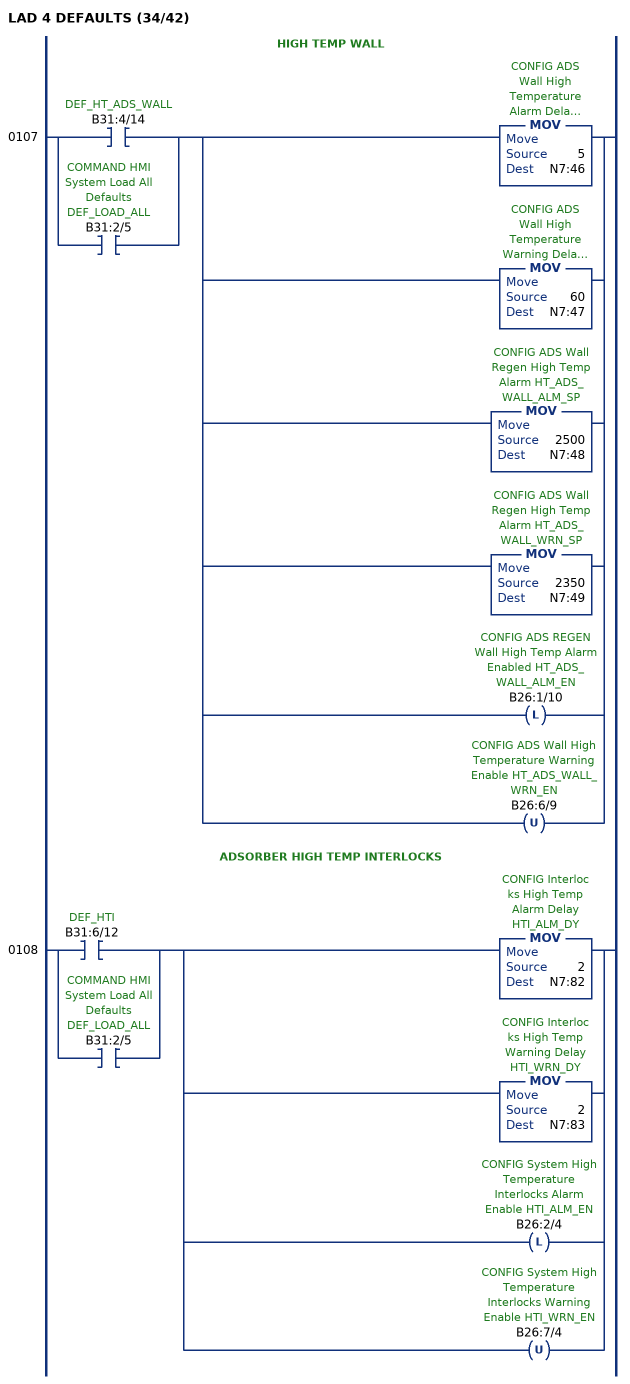
% Rung: 107 %
% TITLE: HIGH TEMP WALL %
SOR BST XIC B31:4/14 NXB XIC B31:2/5 BND BST MOV 5 N7:46 NXB MOV 60 N7:47 NXB MOV 2500 N7:48 NXB MOV 2350 N7:49 NXB OTL B26:1/10 NXB OTU B26:6/9 BND EOR
%   B31:4/14  DEF_HT_ADS_WALL %
%   B31:2/5  DEF_LOAD_ALL  "COMMAND HMI System Load All Defaults" %
%   N7:46  HT_ADS_WALL_ALM_DLY  "CONFIG ADS Wall High Temperature Alarm Delay" %
%   N7:47  HT_ADS_WALL_WRN_DLY  "CONFIG ADS Wall High Temperature Warning Delay" %
%   N7:48  HT_ADS_WALL_ALM_SP  "CONFIG ADS Wall Regen High Temp Alarm" %
%   N7:49  HT_ADS_WALL_WRN_SP  "CONFIG ADS Wall Regen High Temp Alarm" %
%   B26:1/10  HT_ADS_WALL_ALM_EN  "CONFIG ADS REGEN Wall High Temp Alarm Enabled" %
%   B26:6/9  HT_ADS_WALL_WRN_EN  "CONFIG ADS Wall High Temperature Warning Enable" %
% Rung: 108 %
% TITLE: ADSORBER HIGH TEMP INTERLOCKS %
SOR BST XIC B31:6/12 NXB XIC B31:2/5 BND BST MOV 2 N7:82 NXB MOV 2 N7:83 NXB OTL B26:2/4 NXB OTU B26:7/4 BND EOR
%   B31:6/12  DEF_HTI %
%   B31:2/5  DEF_LOAD_ALL  "COMMAND HMI System Load All Defaults" %
%   N7:82  HTI_ALM_DY  "CONFIG Interlocks High Temp Alarm Delay" %
%   N7:83  HTI_WRN_DY  "CONFIG Interlocks High Temp Warning Delay" %
%   B26:2/4  HTI_ALM_EN  "CONFIG System High Temperature Interlocks Alarm Enable" %
%   B26:7/4  HTI_WRN_EN  "CONFIG System High Temperature Interlocks Warning Enable" %

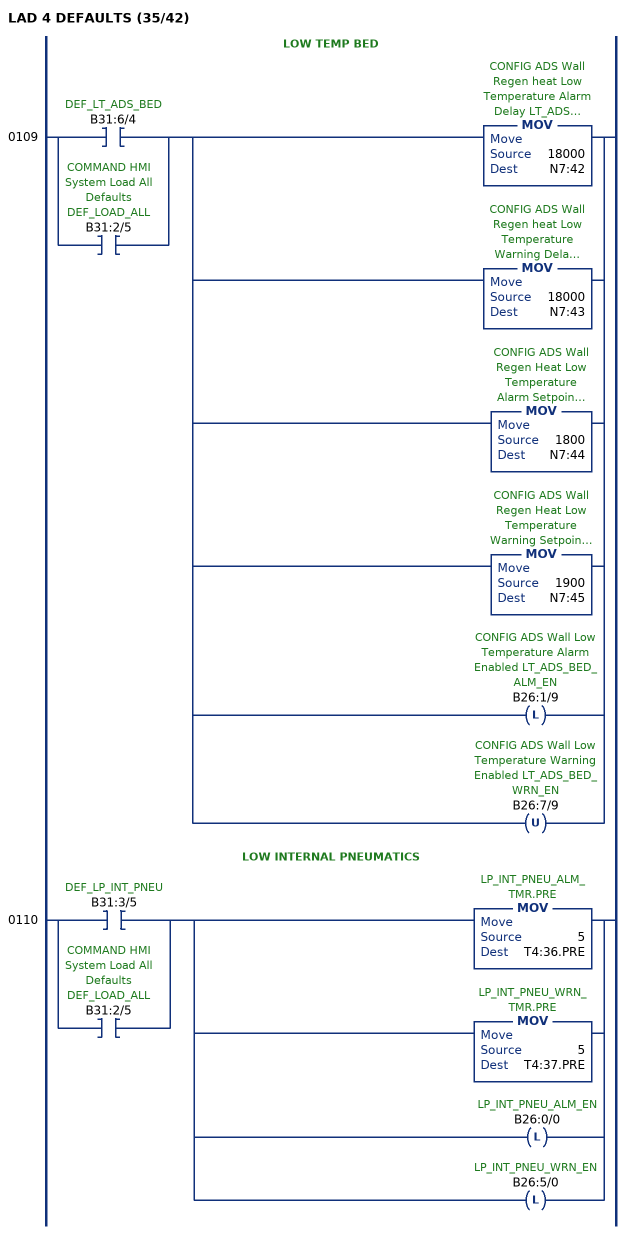
% Rung: 109 %
% TITLE: LOW TEMP BED %
SOR BST XIC B31:6/4 NXB XIC B31:2/5 BND BST MOV 18000 N7:42 NXB MOV 18000 N7:43 NXB MOV 1800 N7:44 NXB MOV 1900 N7:45 NXB OTL B26:1/9 NXB OTU B26:7/9 BND EOR
%   B31:6/4  DEF_LT_ADS_BED %
%   B31:2/5  DEF_LOAD_ALL  "COMMAND HMI System Load All Defaults" %
%   N7:42  LT_ADS_BED_ALM_DLY  "CONFIG ADS Wall Regen heat Low Temperature Alarm Delay" %
%   N7:43  LT_ADS_BED_WRN_DLY  "CONFIG ADS Wall Regen heat Low Temperature Warning Delay" %
%   N7:44  LT_ADS_BED_ALM_SP  "CONFIG ADS Wall Regen Heat Low Temperature Alarm Setpoint" %
%   N7:45  LT_ADS_BED_WRN_SP  "CONFIG ADS Wall Regen Heat Low Temperature Warning Setpoint" %
%   B26:1/9  LT_ADS_BED_ALM_EN  "CONFIG ADS Wall Low Temperature Alarm Enabled" %
%   B26:7/9  LT_ADS_BED_WRN_EN  "CONFIG ADS Wall Low Temperature Warning Enabled" %
% Rung: 110 %
% TITLE: LOW INTERNAL PNEUMATICS %
SOR BST XIC B31:3/5 NXB XIC B31:2/5 BND BST MOV 5 T4:36.PRE NXB MOV 5 T4:37.PRE NXB OTL B26:0/0 NXB OTL B26:5/0 BND EOR
%   B31:3/5  DEF_LP_INT_PNEU %
%   B31:2/5  DEF_LOAD_ALL  "COMMAND HMI System Load All Defaults" %
%   T4:36  LP_INT_PNEU_ALM_TMR %
%   T4:37  LP_INT_PNEU_WRN_TMR %
%   B26:0/0  LP_INT_PNEU_ALM_EN %
%   B26:5/0  LP_INT_PNEU_WRN_EN %

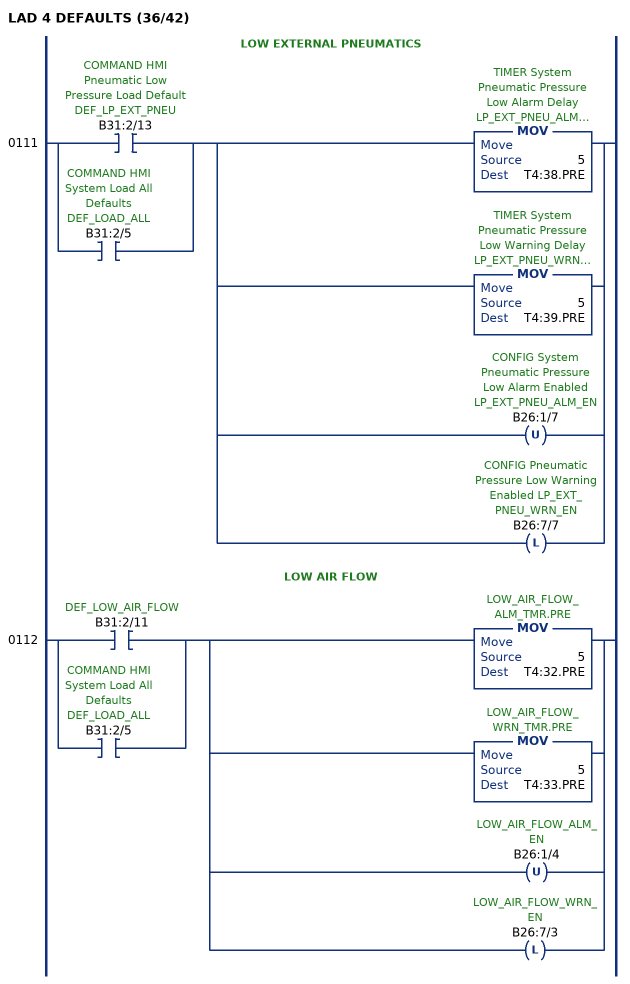
% Rung: 111 %
% TITLE: LOW EXTERNAL PNEUMATICS %
SOR BST XIC B31:2/13 NXB XIC B31:2/5 BND BST MOV 5 T4:38.PRE NXB MOV 5 T4:39.PRE NXB OTU B26:1/7 NXB OTL B26:7/7 BND EOR
%   B31:2/13  DEF_LP_EXT_PNEU  "COMMAND HMI Pneumatic Low Pressure Load Default" %
%   B31:2/5  DEF_LOAD_ALL  "COMMAND HMI System Load All Defaults" %
%   T4:38  LP_EXT_PNEU_ALM_TMR  "TIMER System Pneumatic Pressure Low Alarm Delay" %
%   T4:39  LP_EXT_PNEU_WRN_TMR  "TIMER System Pneumatic Pressure Low Warning Delay" %
%   B26:1/7  LP_EXT_PNEU_ALM_EN  "CONFIG System Pneumatic Pressure Low Alarm Enabled" %
%   B26:7/7  LP_EXT_PNEU_WRN_EN  "CONFIG Pneumatic Pressure Low Warning Enabled" %
% Rung: 112 %
% TITLE: LOW AIR FLOW %
SOR BST XIC B31:2/11 NXB XIC B31:2/5 BND BST MOV 5 T4:32.PRE NXB MOV 5 T4:33.PRE NXB OTU B26:1/4 NXB OTL B26:7/3 BND EOR
%   B31:2/11  DEF_LOW_AIR_FLOW %
%   B31:2/5  DEF_LOAD_ALL  "COMMAND HMI System Load All Defaults" %
%   T4:32  LOW_AIR_FLOW_ALM_TMR %
%   T4:33  LOW_AIR_FLOW_WRN_TMR %
%   B26:1/4  LOW_AIR_FLOW_ALM_EN %
%   B26:7/3  LOW_AIR_FLOW_WRN_EN %

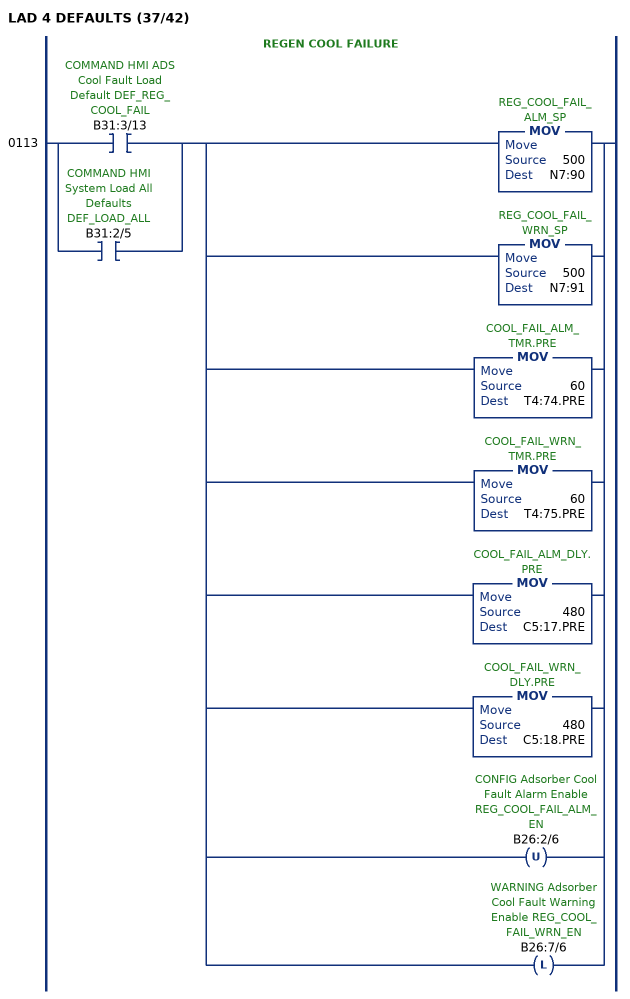
% Rung: 113 %
% TITLE: REGEN COOL FAILURE %
SOR BST XIC B31:3/13 NXB XIC B31:2/5 BND BST MOV 500 N7:90 NXB MOV 500 N7:91 NXB MOV 60 T4:74.PRE NXB MOV 60 T4:75.PRE NXB MOV 480 C5:17.PRE NXB MOV 480 C5:18.PRE NXB OTU B26:2/6 NXB OTL B26:7/6 BND EOR
%   B31:3/13  DEF_REG_COOL_FAIL  "COMMAND HMI ADS Cool Fault Load Default" %
%   B31:2/5  DEF_LOAD_ALL  "COMMAND HMI System Load All Defaults" %
%   N7:90  REG_COOL_FAIL_ALM_SP %
%   N7:91  REG_COOL_FAIL_WRN_SP %
%   T4:74  COOL_FAIL_ALM_TMR %
%   T4:75  COOL_FAIL_WRN_TMR %
%   C5:17  COOL_FAIL_ALM_DLY %
%   C5:18  COOL_FAIL_WRN_DLY %
%   B26:2/6  REG_COOL_FAIL_ALM_EN  "CONFIG Adsorber Cool Fault Alarm Enable" %
%   B26:7/6  REG_COOL_FAIL_WRN_EN  "WARNING Adsorber Cool Fault Warning Enable" %

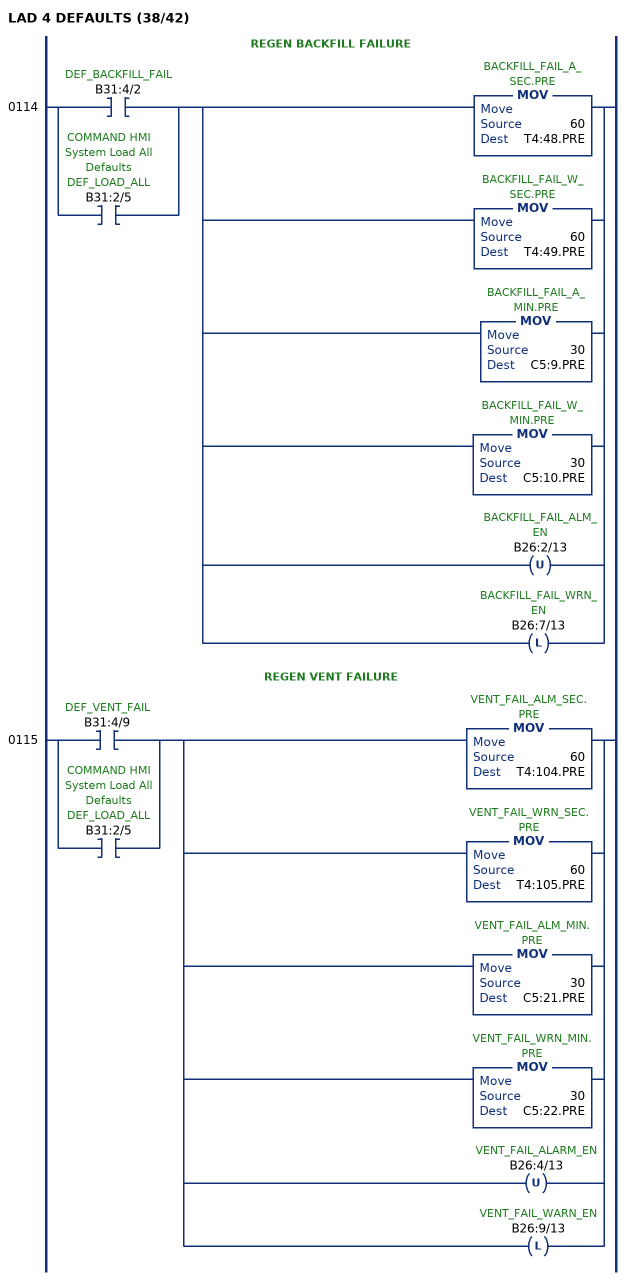
% Rung: 114 %
% TITLE: REGEN BACKFILL FAILURE %
SOR BST XIC B31:4/2 NXB XIC B31:2/5 BND BST MOV 60 T4:48.PRE NXB MOV 60 T4:49.PRE NXB MOV 30 C5:9.PRE NXB MOV 30 C5:10.PRE NXB OTU B26:2/13 NXB OTL B26:7/13 BND EOR
%   B31:4/2  DEF_BACKFILL_FAIL %
%   B31:2/5  DEF_LOAD_ALL  "COMMAND HMI System Load All Defaults" %
%   T4:48  BACKFILL_FAIL_A_SEC %
%   T4:49  BACKFILL_FAIL_W_SEC %
%   C5:9  BACKFILL_FAIL_A_MIN %
%   C5:10  BACKFILL_FAIL_W_MIN %
%   B26:2/13  BACKFILL_FAIL_ALM_EN %
%   B26:7/13  BACKFILL_FAIL_WRN_EN %
% Rung: 115 %
% TITLE: REGEN VENT FAILURE %
SOR BST XIC B31:4/9 NXB XIC B31:2/5 BND BST MOV 60 T4:104.PRE NXB MOV 60 T4:105.PRE NXB MOV 30 C5:21.PRE NXB MOV 30 C5:22.PRE NXB OTU B26:4/13 NXB OTL B26:9/13 BND EOR
%   B31:4/9  DEF_VENT_FAIL %
%   B31:2/5  DEF_LOAD_ALL  "COMMAND HMI System Load All Defaults" %
%   T4:104  VENT_FAIL_ALM_SEC %
%   T4:105  VENT_FAIL_WRN_SEC %
%   C5:21  VENT_FAIL_ALM_MIN %
%   C5:22  VENT_FAIL_WRN_MIN %
%   B26:4/13  VENT_FAIL_ALARM_EN %
%   B26:9/13  VENT_FAIL_WARN_EN %

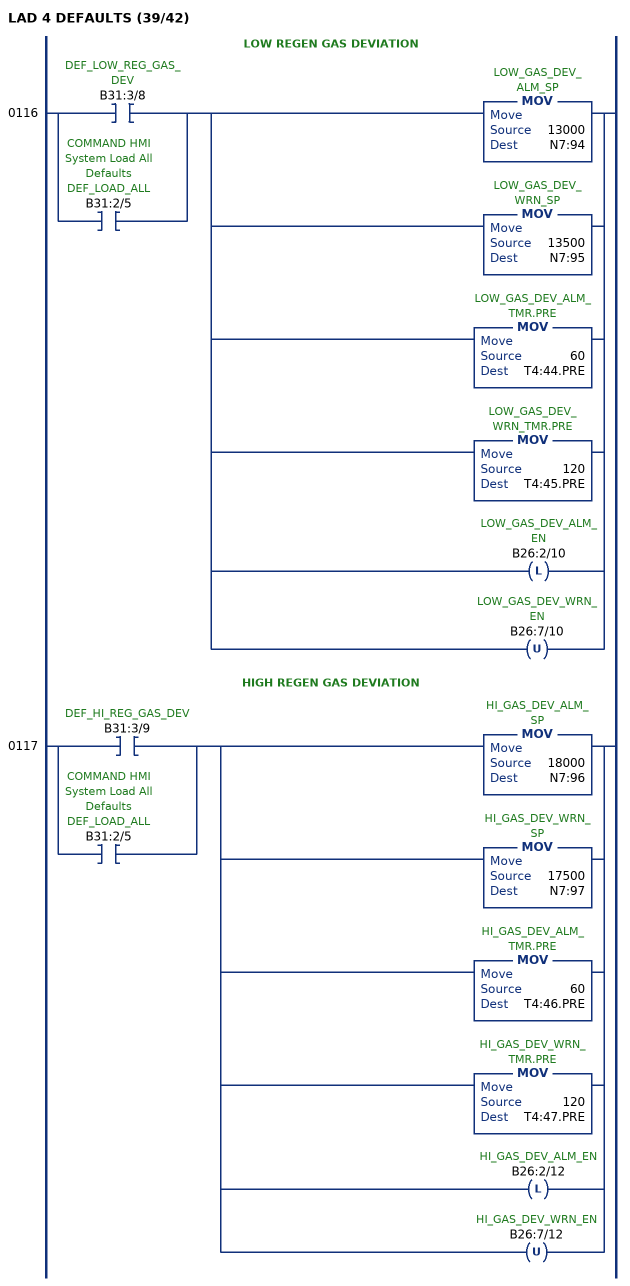
% Rung: 116 %
% TITLE: LOW REGEN GAS DEVIATION %
SOR BST XIC B31:3/8 NXB XIC B31:2/5 BND BST MOV 13000 N7:94 NXB MOV 13500 N7:95 NXB MOV 60 T4:44.PRE NXB MOV 120 T4:45.PRE NXB OTL B26:2/10 NXB OTU B26:7/10 BND EOR
%   B31:3/8  DEF_LOW_REG_GAS_DEV %
%   B31:2/5  DEF_LOAD_ALL  "COMMAND HMI System Load All Defaults" %
%   N7:94  LOW_GAS_DEV_ALM_SP %
%   N7:95  LOW_GAS_DEV_WRN_SP %
%   T4:44  LOW_GAS_DEV_ALM_TMR %
%   T4:45  LOW_GAS_DEV_WRN_TMR %
%   B26:2/10  LOW_GAS_DEV_ALM_EN %
%   B26:7/10  LOW_GAS_DEV_WRN_EN %
% Rung: 117 %
% TITLE: HIGH REGEN GAS DEVIATION %
SOR BST XIC B31:3/9 NXB XIC B31:2/5 BND BST MOV 18000 N7:96 NXB MOV 17500 N7:97 NXB MOV 60 T4:46.PRE NXB MOV 120 T4:47.PRE NXB OTL B26:2/12 NXB OTU B26:7/12 BND EOR
%   B31:3/9  DEF_HI_REG_GAS_DEV %
%   B31:2/5  DEF_LOAD_ALL  "COMMAND HMI System Load All Defaults" %
%   N7:96  HI_GAS_DEV_ALM_SP %
%   N7:97  HI_GAS_DEV_WRN_SP %
%   T4:46  HI_GAS_DEV_ALM_TMR %
%   T4:47  HI_GAS_DEV_WRN_TMR %
%   B26:2/12  HI_GAS_DEV_ALM_EN %
%   B26:7/12  HI_GAS_DEV_WRN_EN %

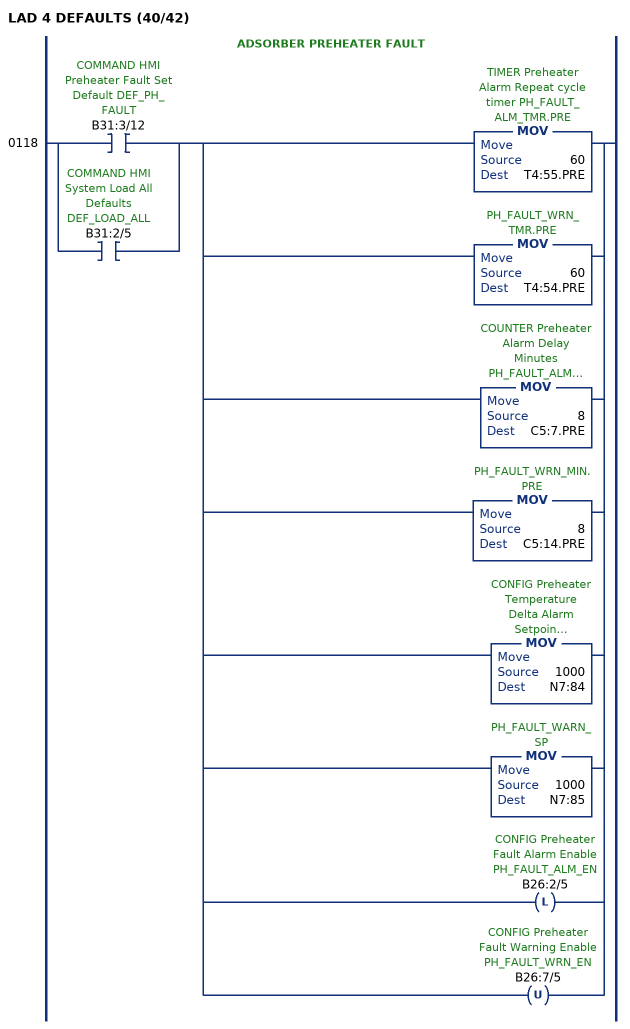
% Rung: 118 %
% TITLE: ADSORBER PREHEATER FAULT %
SOR BST XIC B31:3/12 NXB XIC B31:2/5 BND BST MOV 60 T4:55.PRE NXB MOV 60 T4:54.PRE NXB MOV 8 C5:7.PRE NXB MOV 8 C5:14.PRE NXB MOV 1000 N7:84 NXB MOV 1000 N7:85 NXB OTL B26:2/5 NXB OTU B26:7/5 BND EOR
%   B31:3/12  DEF_PH_FAULT  "COMMAND HMI Preheater Fault Set Default" %
%   B31:2/5  DEF_LOAD_ALL  "COMMAND HMI System Load All Defaults" %
%   T4:55  PH_FAULT_ALM_TMR  "TIMER Preheater Alarm Repeat cycle timer" %
%   T4:54  PH_FAULT_WRN_TMR %
%   C5:7  PH_FAULT_ALM_MIN  "COUNTER Preheater Alarm Delay Minutes" %
%   C5:14  PH_FAULT_WRN_MIN %
%   N7:84  PH_FAULT_ALARM_SP  "CONFIG Preheater Temperature Delta Alarm Setpoint" %
%   N7:85  PH_FAULT_WARN_SP %
%   B26:2/5  PH_FAULT_ALM_EN  "CONFIG Preheater Fault Alarm Enable" %
%   B26:7/5  PH_FAULT_WRN_EN  "CONFIG Preheater Fault Warning Enable" %

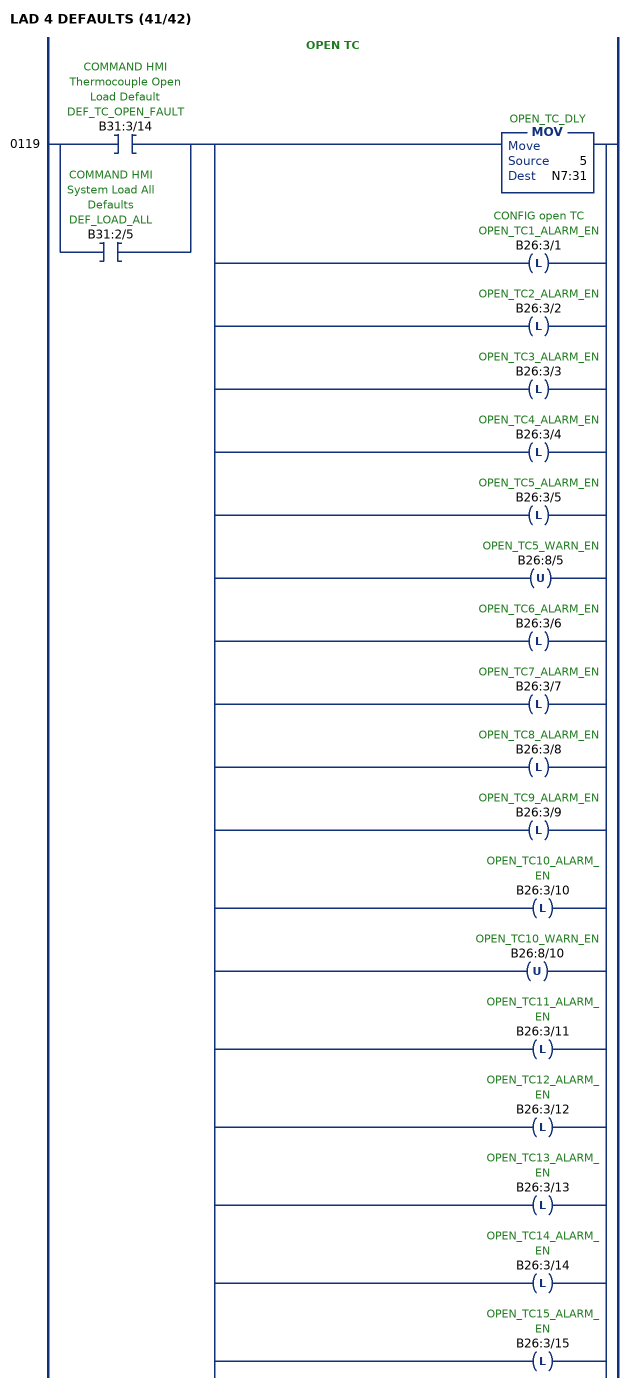

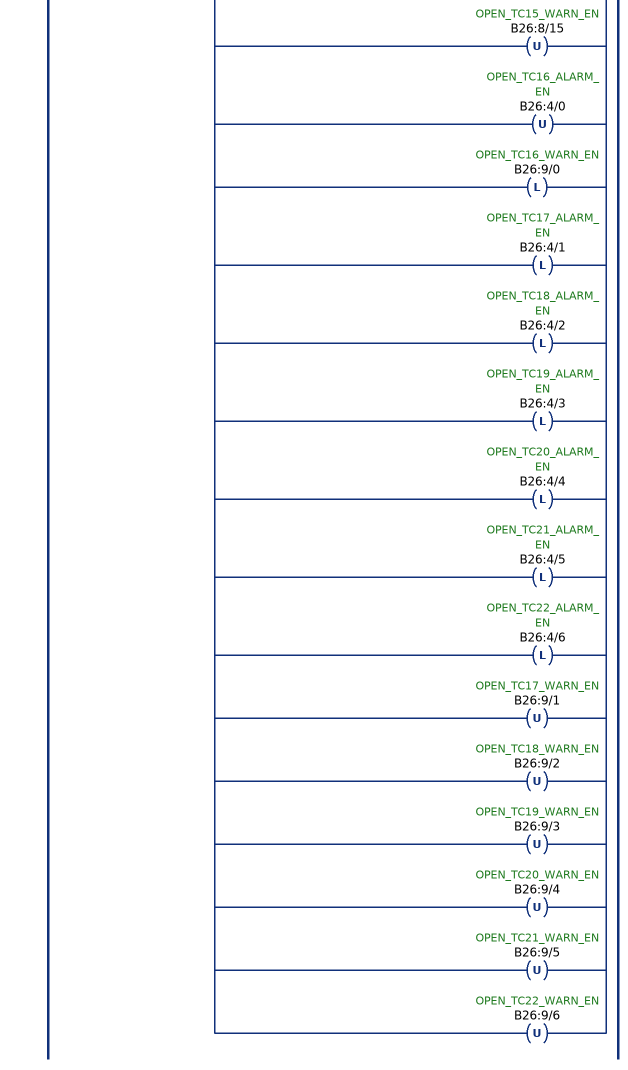
% Rung: 119 %
% TITLE: OPEN TC %
SOR BST XIC B31:3/14 NXB XIC B31:2/5 BND BST MOV 5 N7:31 NXB BST OTL B26:3/1 NXB OTL B26:3/2 NXB OTL B26:3/3 NXB OTL B26:3/4 NXB OTL B26:3/5 NXB OTU B26:8/5 BND NXB BST OTL B26:3/6 NXB OTL B26:3/7 NXB OTL B26:3/8 NXB OTL B26:3/9 NXB OTL B26:3/10 NXB OTU B26:8/10 BND NXB BST OTL B26:3/11 NXB OTL B26:3/12 NXB OTL B26:3/13 NXB OTL B26:3/14 NXB OTL B26:3/15 NXB OTU B26:8/15 BND NXB BST OTU B26:4/0 NXB OTL B26:9/0 BND NXB BST OTL B26:4/1 NXB OTL B26:4/2 NXB OTL B26:4/3 NXB OTL B26:4/4 NXB OTL B26:4/5 NXB OTL B26:4/6 BND NXB BST OTU B26:9/1 NXB OTU B26:9/2 NXB OTU B26:9/3 NXB OTU B26:9/4 NXB OTU B26:9/5 NXB OTU B26:9/6 BND BND EOR
%   B31:3/14  DEF_TC_OPEN_FAULT  "COMMAND HMI Thermocouple Open Load Default" %
%   B31:2/5  DEF_LOAD_ALL  "COMMAND HMI System Load All Defaults" %
%   N7:31  OPEN_TC_DLY %
%   B26:3/1  OPEN_TC1_ALARM_EN  "CONFIG open TC" %
%   B26:3/2  OPEN_TC2_ALARM_EN %
%   B26:3/3  OPEN_TC3_ALARM_EN %
%   B26:3/4  OPEN_TC4_ALARM_EN %
%   B26:3/5  OPEN_TC5_ALARM_EN %
%   B26:8/5  OPEN_TC5_WARN_EN %
%   B26:3/6  OPEN_TC6_ALARM_EN %
%   B26:3/7  OPEN_TC7_ALARM_EN %
%   B26:3/8  OPEN_TC8_ALARM_EN %
%   B26:3/9  OPEN_TC9_ALARM_EN %
%   B26:3/10  OPEN_TC10_ALARM_EN %
%   B26:8/10  OPEN_TC10_WARN_EN %
%   B26:3/11  OPEN_TC11_ALARM_EN %
%   B26:3/12  OPEN_TC12_ALARM_EN %
%   B26:3/13  OPEN_TC13_ALARM_EN %
%   B26:3/14  OPEN_TC14_ALARM_EN %
%   B26:3/15  OPEN_TC15_ALARM_EN %
%   B26:8/15  OPEN_TC15_WARN_EN %
%   B26:4/0  OPEN_TC16_ALARM_EN %
%   B26:9/0  OPEN_TC16_WARN_EN %
%   B26:4/1  OPEN_TC17_ALARM_EN %
%   B26:4/2  OPEN_TC18_ALARM_EN %
%   B26:4/3  OPEN_TC19_ALARM_EN %
%   B26:4/4  OPEN_TC20_ALARM_EN %
%   B26:4/5  OPEN_TC21_ALARM_EN %
%   B26:4/6  OPEN_TC22_ALARM_EN %
%   B26:9/1  OPEN_TC17_WARN_EN %
%   B26:9/2  OPEN_TC18_WARN_EN %
%   B26:9/3  OPEN_TC19_WARN_EN %
%   B26:9/4  OPEN_TC20_WARN_EN %
%   B26:9/5  OPEN_TC21_WARN_EN %
%   B26:9/6  OPEN_TC22_WARN_EN %

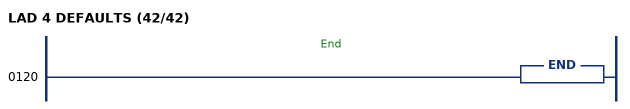
% Rung: 120 %
% End %
SOR END EOR

LADDER 5 "SYS_FAULTS"    % Monitors the system fault conditions %
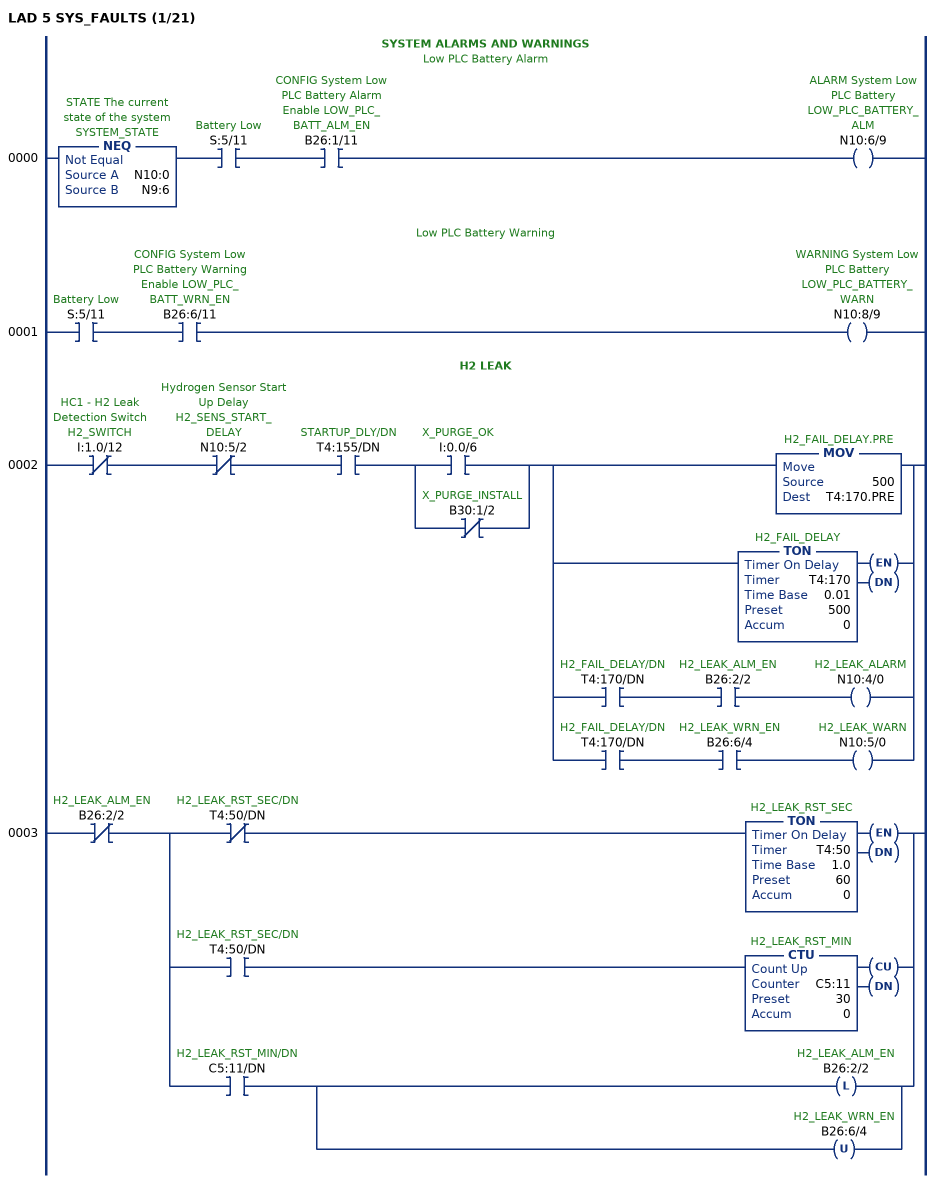
% Rung: 0 %
% TITLE: SYSTEM ALARMS AND WARNINGS %
% Low PLC Battery Alarm %
SOR NEQ N10:0 N9:6 XIC S:5/11 XIC B26:1/11 OTE N10:6/9 EOR
%   N10:0  SYSTEM_STATE  "STATE The current state of the system" %
%   N9:6  SYSTEM_PURGE %
%   S:5/11  "Battery Low" %
%   B26:1/11  LOW_PLC_BATT_ALM_EN  "CONFIG System Low PLC Battery Alarm Enable" %
%   N10:6/9  LOW_PLC_BATTERY_ALM  "ALARM System Low PLC Battery" %
% Rung: 1 %
% Low PLC Battery Warning %
SOR XIC S:5/11 XIC B26:6/11 OTE N10:8/9 EOR
%   S:5/11  "Battery Low" %
%   B26:6/11  LOW_PLC_BATT_WRN_EN  "CONFIG System Low PLC Battery Warning Enable" %
%   N10:8/9  LOW_PLC_BATTERY_WARN  "WARNING System Low PLC Battery" %
% Rung: 2 %
% TITLE: H2 LEAK %
SOR XIO I:1.0/12 XIO N10:5/2 XIC T4:155/DN BST XIC I:0.0/6 NXB XIO B30:1/2 BND BST MOV 500 T4:170.PRE NXB TON T4:170 0.01 500 0 NXB XIC T4:170/DN XIC B26:2/2 OTE N10:4/0 NXB XIC T4:170/DN XIC B26:6/4 OTE N10:5/0 BND EOR
%   I:1.0/12  H2_SWITCH  "HC1 - H2 Leak Detection Switch" %
%   N10:5/2  H2_SENS_START_DELAY  "Hydrogen Sensor Start Up Delay" %
%   T4:155  STARTUP_DLY %
%   I:0.0/6  X_PURGE_OK %
%   B30:1/2  X_PURGE_INSTALL %
%   T4:170  H2_FAIL_DELAY %
%   B26:2/2  H2_LEAK_ALM_EN %
%   N10:4/0  H2_LEAK_ALARM %
%   B26:6/4  H2_LEAK_WRN_EN %
%   N10:5/0  H2_LEAK_WARN %
% Rung: 3 %
SOR XIO B26:2/2 BST XIO T4:50/DN TON T4:50 1.0 60 0 NXB XIC T4:50/DN CTU C5:11 30 0 NXB XIC C5:11/DN BST OTL B26:2/2 NXB OTU B26:6/4 BND BND EOR
%   B26:2/2  H2_LEAK_ALM_EN %
%   T4:50  H2_LEAK_RST_SEC %
%   C5:11  H2_LEAK_RST_MIN %
%   B26:6/4  H2_LEAK_WRN_EN %

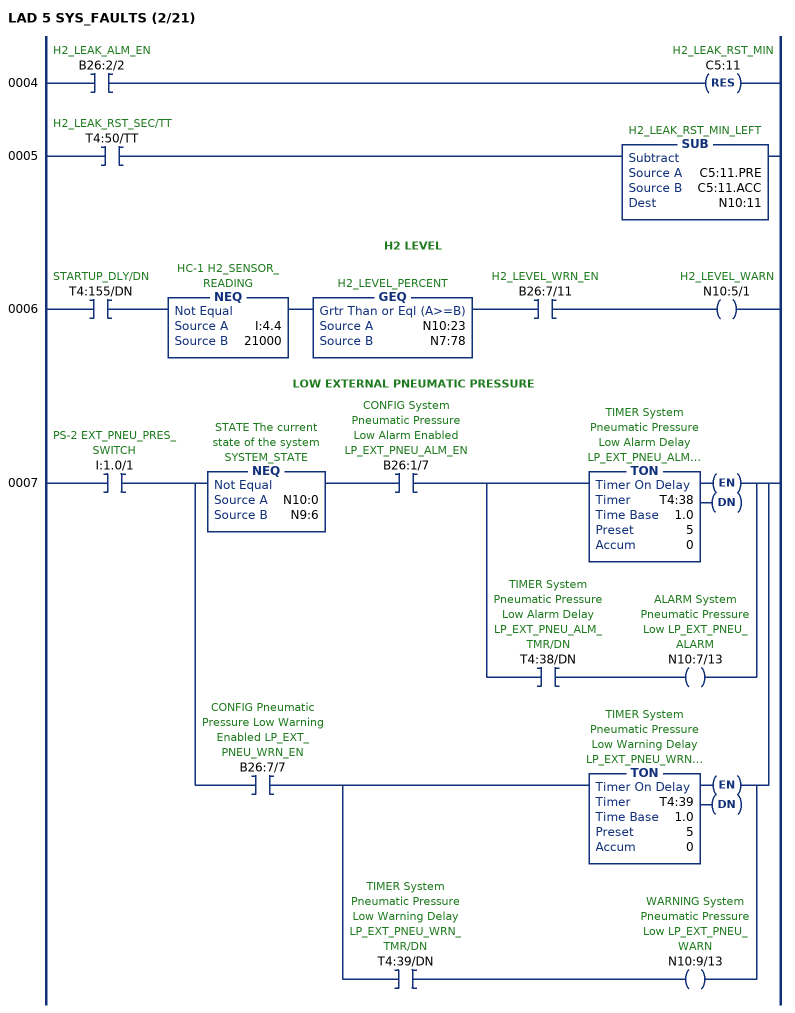
% Rung: 4 %
SOR XIC B26:2/2 RES C5:11 EOR
%   B26:2/2  H2_LEAK_ALM_EN %
%   C5:11  H2_LEAK_RST_MIN %
% Rung: 5 %
SOR XIC T4:50/TT SUB C5:11.PRE C5:11.ACC N10:11 EOR
%   T4:50  H2_LEAK_RST_SEC %
%   C5:11  H2_LEAK_RST_MIN %
%   N10:11  H2_LEAK_RST_MIN_LEFT %
% Rung: 6 %
% TITLE: H2 LEVEL %
SOR XIC T4:155/DN NEQ I:4.4 21000 GEQ N10:23 N7:78 XIC B26:7/11 OTE N10:5/1 EOR
%   T4:155  STARTUP_DLY %
%   I:4.4  H2_SENSOR_READING  "HC-1" %
%   N10:23  H2_LEVEL_PERCENT %
%   N7:78  H2_LEVEL_WRN_SP %
%   B26:7/11  H2_LEVEL_WRN_EN %
%   N10:5/1  H2_LEVEL_WARN %
% Rung: 7 %
% TITLE: LOW EXTERNAL PNEUMATIC PRESSURE %
SOR XIC I:1.0/1 BST NEQ N10:0 N9:6 XIC B26:1/7 BST TON T4:38 1.0 5 0 NXB XIC T4:38/DN OTE N10:7/13 BND NXB XIC B26:7/7 BST TON T4:39 1.0 5 0 NXB XIC T4:39/DN OTE N10:9/13 BND BND EOR
%   I:1.0/1  EXT_PNEU_PRES_SWITCH  "PS-2" %
%   N10:0  SYSTEM_STATE  "STATE The current state of the system" %
%   N9:6  SYSTEM_PURGE %
%   B26:1/7  LP_EXT_PNEU_ALM_EN  "CONFIG System Pneumatic Pressure Low Alarm Enabled" %
%   T4:38  LP_EXT_PNEU_ALM_TMR  "TIMER System Pneumatic Pressure Low Alarm Delay" %
%   N10:7/13  LP_EXT_PNEU_ALARM  "ALARM System Pneumatic Pressure Low" %
%   B26:7/7  LP_EXT_PNEU_WRN_EN  "CONFIG Pneumatic Pressure Low Warning Enabled" %
%   T4:39  LP_EXT_PNEU_WRN_TMR  "TIMER System Pneumatic Pressure Low Warning Delay" %
%   N10:9/13  LP_EXT_PNEU_WARN  "WARNING System Pneumatic Pressure Low" %

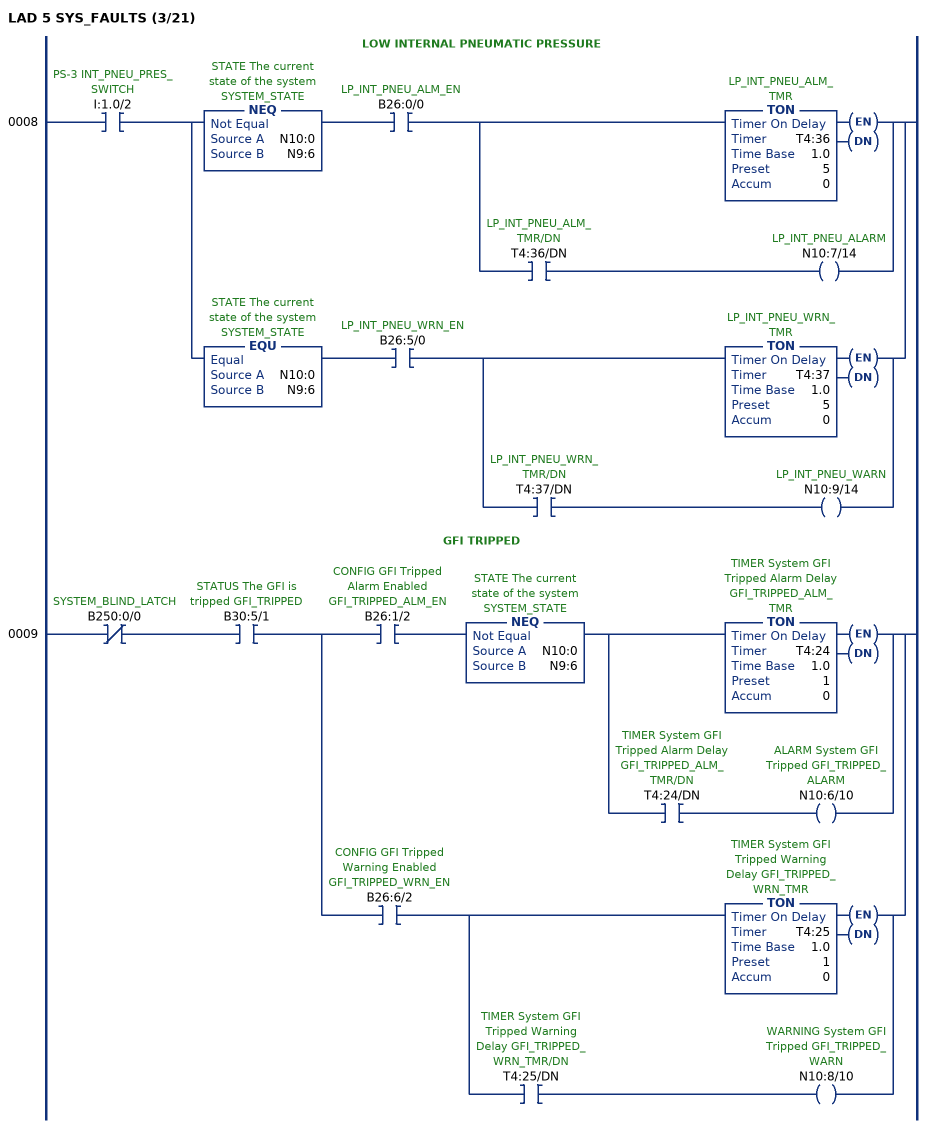
% Rung: 8 %
% TITLE: LOW INTERNAL PNEUMATIC PRESSURE %
SOR XIC I:1.0/2 BST NEQ N10:0 N9:6 XIC B26:0/0 BST TON T4:36 1.0 5 0 NXB XIC T4:36/DN OTE N10:7/14 BND NXB EQU N10:0 N9:6 XIC B26:5/0 BST TON T4:37 1.0 5 0 NXB XIC T4:37/DN OTE N10:9/14 BND BND EOR
%   I:1.0/2  INT_PNEU_PRES_SWITCH  "PS-3" %
%   N10:0  SYSTEM_STATE  "STATE The current state of the system" %
%   N9:6  SYSTEM_PURGE %
%   B26:0/0  LP_INT_PNEU_ALM_EN %
%   T4:36  LP_INT_PNEU_ALM_TMR %
%   N10:7/14  LP_INT_PNEU_ALARM %
%   B26:5/0  LP_INT_PNEU_WRN_EN %
%   T4:37  LP_INT_PNEU_WRN_TMR %
%   N10:9/14  LP_INT_PNEU_WARN %
% Rung: 9 %
% TITLE: GFI TRIPPED %
SOR XIO B250:0/0 XIC B30:5/1 BST XIC B26:1/2 NEQ N10:0 N9:6 BST TON T4:24 1.0 1 0 NXB XIC T4:24/DN OTE N10:6/10 BND NXB XIC B26:6/2 BST TON T4:25 1.0 1 0 NXB XIC T4:25/DN OTE N10:8/10 BND BND EOR
%   B250:0/0  SYSTEM_BLIND_LATCH %
%   B30:5/1  GFI_TRIPPED  "STATUS The GFI is tripped" %
%   B26:1/2  GFI_TRIPPED_ALM_EN  "CONFIG GFI Tripped Alarm Enabled" %
%   N10:0  SYSTEM_STATE  "STATE The current state of the system" %
%   N9:6  SYSTEM_PURGE %
%   T4:24  GFI_TRIPPED_ALM_TMR  "TIMER System GFI Tripped Alarm Delay" %
%   N10:6/10  GFI_TRIPPED_ALARM  "ALARM System GFI Tripped" %
%   B26:6/2  GFI_TRIPPED_WRN_EN  "CONFIG GFI Tripped Warning Enabled" %
%   T4:25  GFI_TRIPPED_WRN_TMR  "TIMER System GFI Tripped Warning Delay" %
%   N10:8/10  GFI_TRIPPED_WARN  "WARNING System GFI Tripped" %

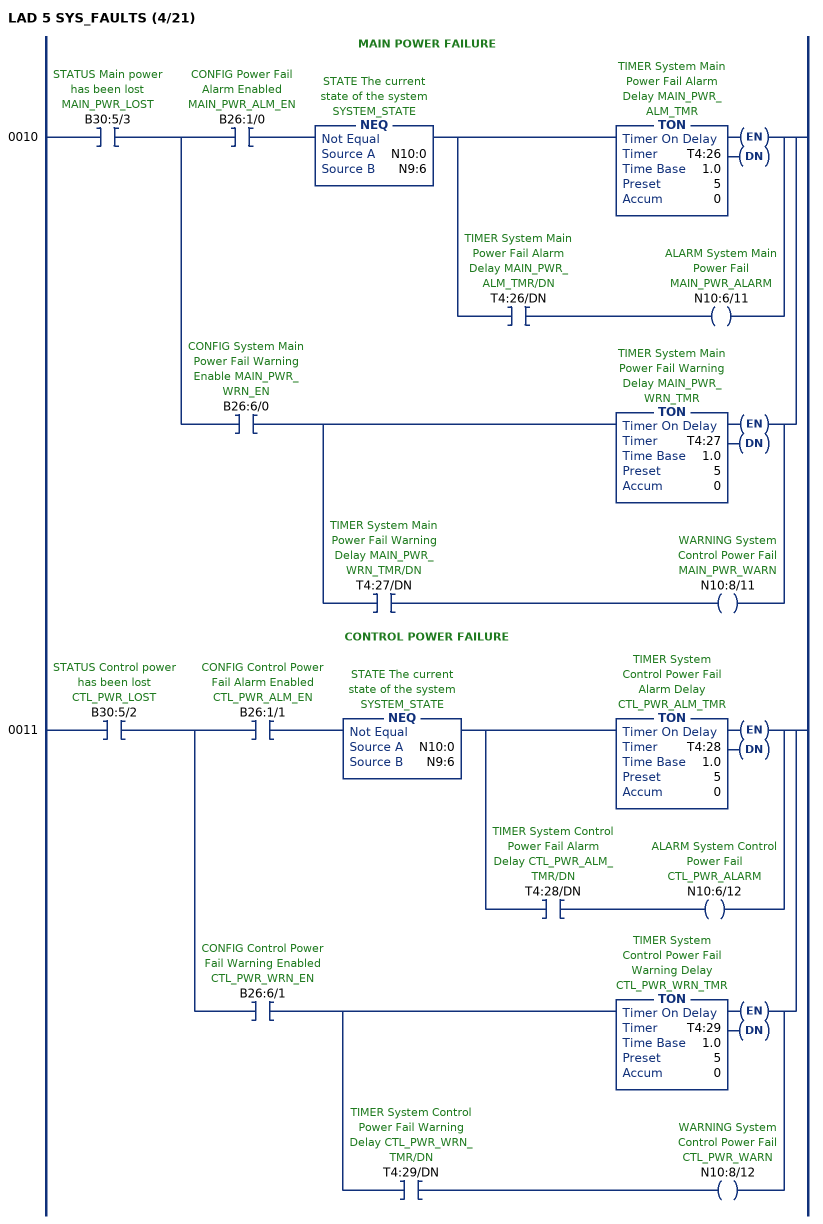
% Rung: 10 %
% TITLE: MAIN POWER FAILURE %
SOR XIC B30:5/3 BST XIC B26:1/0 NEQ N10:0 N9:6 BST TON T4:26 1.0 5 0 NXB XIC T4:26/DN OTE N10:6/11 BND NXB XIC B26:6/0 BST TON T4:27 1.0 5 0 NXB XIC T4:27/DN OTE N10:8/11 BND BND EOR
%   B30:5/3  MAIN_PWR_LOST  "STATUS Main power has been lost" %
%   B26:1/0  MAIN_PWR_ALM_EN  "CONFIG Power Fail Alarm Enabled" %
%   N10:0  SYSTEM_STATE  "STATE The current state of the system" %
%   N9:6  SYSTEM_PURGE %
%   T4:26  MAIN_PWR_ALM_TMR  "TIMER System Main Power Fail Alarm Delay" %
%   N10:6/11  MAIN_PWR_ALARM  "ALARM System Main Power Fail" %
%   B26:6/0  MAIN_PWR_WRN_EN  "CONFIG System Main Power Fail Warning Enable" %
%   T4:27  MAIN_PWR_WRN_TMR  "TIMER System Main Power Fail Warning Delay" %
%   N10:8/11  MAIN_PWR_WARN  "WARNING System Control Power Fail" %
% Rung: 11 %
% TITLE: CONTROL POWER FAILURE %
SOR XIC B30:5/2 BST XIC B26:1/1 NEQ N10:0 N9:6 BST TON T4:28 1.0 5 0 NXB XIC T4:28/DN OTE N10:6/12 BND NXB XIC B26:6/1 BST TON T4:29 1.0 5 0 NXB XIC T4:29/DN OTE N10:8/12 BND BND EOR
%   B30:5/2  CTL_PWR_LOST  "STATUS Control power has been lost" %
%   B26:1/1  CTL_PWR_ALM_EN  "CONFIG Control Power Fail Alarm Enabled" %
%   N10:0  SYSTEM_STATE  "STATE The current state of the system" %
%   N9:6  SYSTEM_PURGE %
%   T4:28  CTL_PWR_ALM_TMR  "TIMER System Control Power Fail Alarm Delay" %
%   N10:6/12  CTL_PWR_ALARM  "ALARM System Control Power Fail" %
%   B26:6/1  CTL_PWR_WRN_EN  "CONFIG Control Power Fail Warning Enabled" %
%   T4:29  CTL_PWR_WRN_TMR  "TIMER System Control Power Fail Warning Delay" %
%   N10:8/12  CTL_PWR_WARN  "WARNING System Control Power Fail" %

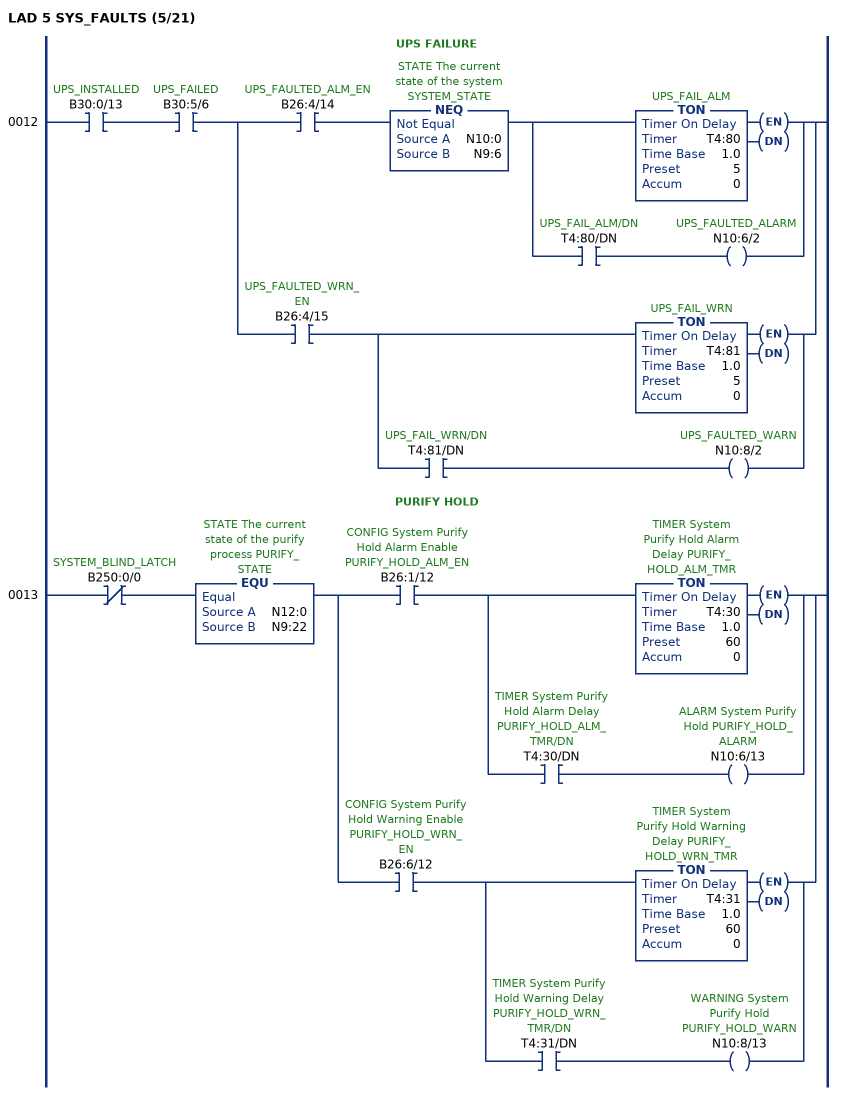
% Rung: 12 %
% TITLE: UPS FAILURE %
SOR XIC B30:0/13 XIC B30:5/6 BST XIC B26:4/14 NEQ N10:0 N9:6 BST TON T4:80 1.0 5 0 NXB XIC T4:80/DN OTE N10:6/2 BND NXB XIC B26:4/15 BST TON T4:81 1.0 5 0 NXB XIC T4:81/DN OTE N10:8/2 BND BND EOR
%   B30:0/13  UPS_INSTALLED %
%   B30:5/6  UPS_FAILED %
%   B26:4/14  UPS_FAULTED_ALM_EN %
%   N10:0  SYSTEM_STATE  "STATE The current state of the system" %
%   N9:6  SYSTEM_PURGE %
%   T4:80  UPS_FAIL_ALM %
%   N10:6/2  UPS_FAULTED_ALARM %
%   B26:4/15  UPS_FAULTED_WRN_EN %
%   T4:81  UPS_FAIL_WRN %
%   N10:8/2  UPS_FAULTED_WARN %
% Rung: 13 %
% TITLE: PURIFY HOLD %
SOR XIO B250:0/0 EQU N12:0 N9:22 BST XIC B26:1/12 BST TON T4:30 1.0 60 0 NXB XIC T4:30/DN OTE N10:6/13 BND NXB XIC B26:6/12 BST TON T4:31 1.0 60 0 NXB XIC T4:31/DN OTE N10:8/13 BND BND EOR
%   B250:0/0  SYSTEM_BLIND_LATCH %
%   N12:0  PURIFY_STATE  "STATE The current state of the purify process" %
%   N9:22  PURIFY_HOLD  "STATE Purify Hold" %
%   B26:1/12  PURIFY_HOLD_ALM_EN  "CONFIG System Purify Hold Alarm Enable" %
%   T4:30  PURIFY_HOLD_ALM_TMR  "TIMER System Purify Hold Alarm Delay" %
%   N10:6/13  PURIFY_HOLD_ALARM  "ALARM System Purify Hold" %
%   B26:6/12  PURIFY_HOLD_WRN_EN  "CONFIG System Purify Hold Warning Enable" %
%   T4:31  PURIFY_HOLD_WRN_TMR  "TIMER System Purify Hold Warning Delay" %
%   N10:8/13  PURIFY_HOLD_WARN  "WARNING System Purify Hold" %

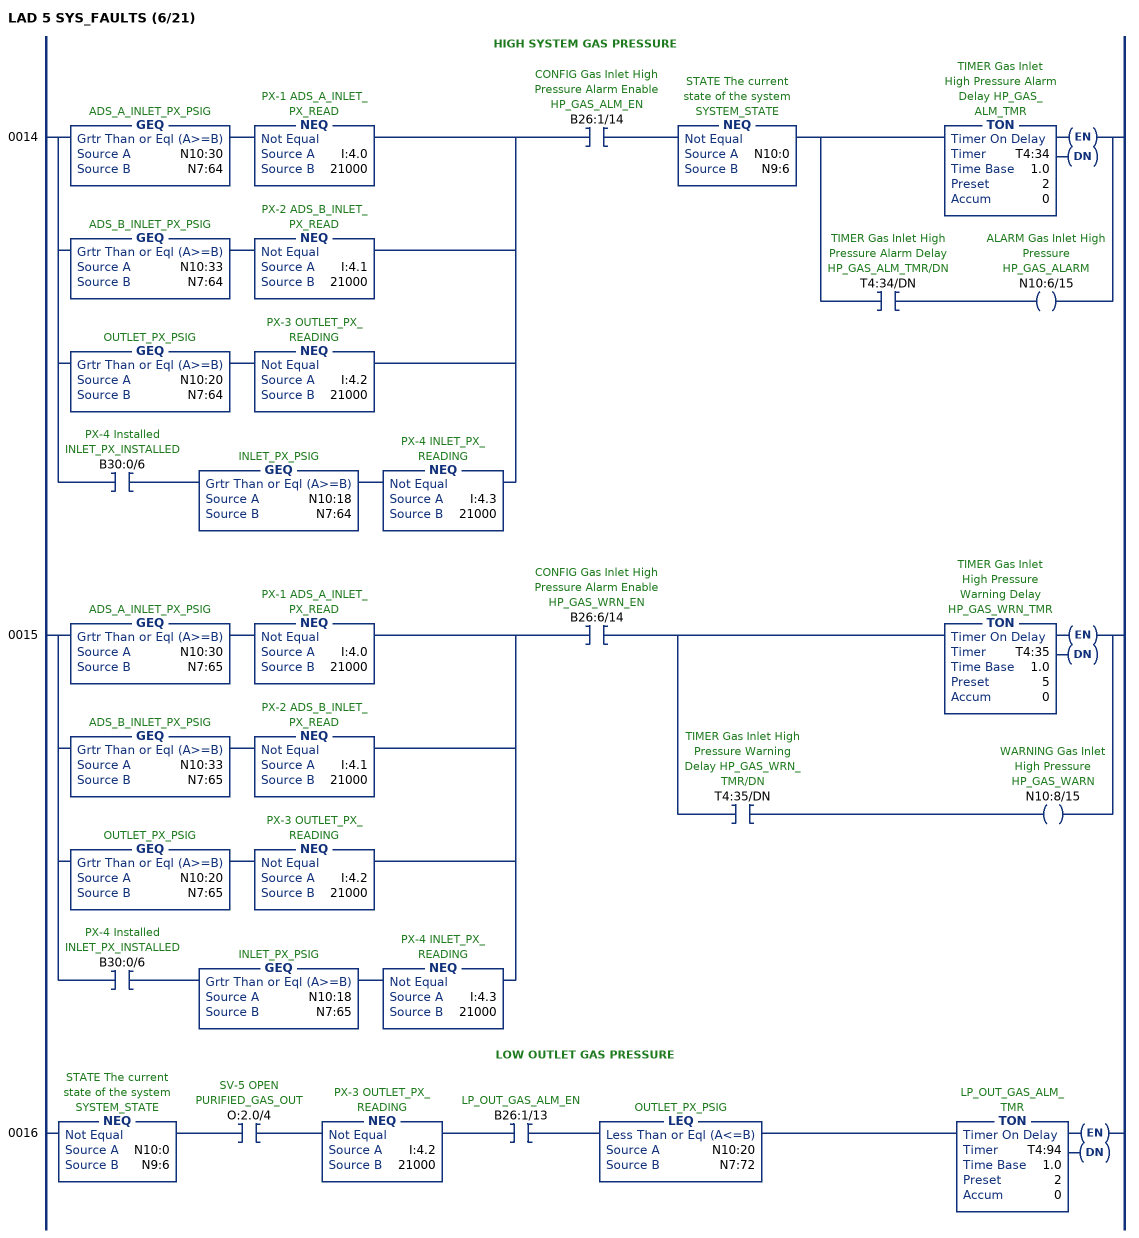
% Rung: 14 %
% TITLE: HIGH SYSTEM GAS PRESSURE %
SOR BST GEQ N10:30 N7:64 NEQ I:4.0 21000 NXB GEQ N10:33 N7:64 NEQ I:4.1 21000 NXB GEQ N10:20 N7:64 NEQ I:4.2 21000 NXB XIC B30:0/6 GEQ N10:18 N7:64 NEQ I:4.3 21000 BND XIC B26:1/14 NEQ N10:0 N9:6 BST TON T4:34 1.0 2 0 NXB XIC T4:34/DN OTE N10:6/15 BND EOR
%   N10:30  ADS_A_INLET_PX_PSIG %
%   N7:64  HP_GAS_ALM_SP  "CONFIG Gas Inlet High Pressure Alarm Setpoint" %
%   I:4.0  ADS_A_INLET_PX_READ  "PX-1" %
%   N10:33  ADS_B_INLET_PX_PSIG %
%   I:4.1  ADS_B_INLET_PX_READ  "PX-2" %
%   N10:20  OUTLET_PX_PSIG %
%   I:4.2  OUTLET_PX_READING  "PX-3" %
%   B30:0/6  INLET_PX_INSTALLED  "PX-4 Installed" %
%   N10:18  INLET_PX_PSIG %
%   I:4.3  INLET_PX_READING  "PX-4" %
%   B26:1/14  HP_GAS_ALM_EN  "CONFIG Gas Inlet High Pressure Alarm Enable" %
%   N10:0  SYSTEM_STATE  "STATE The current state of the system" %
%   N9:6  SYSTEM_PURGE %
%   T4:34  HP_GAS_ALM_TMR  "TIMER Gas Inlet High Pressure Alarm Delay" %
%   N10:6/15  HP_GAS_ALARM  "ALARM Gas Inlet High Pressure" %
% Rung: 15 %
SOR BST GEQ N10:30 N7:65 NEQ I:4.0 21000 NXB GEQ N10:33 N7:65 NEQ I:4.1 21000 NXB GEQ N10:20 N7:65 NEQ I:4.2 21000 NXB XIC B30:0/6 GEQ N10:18 N7:65 NEQ I:4.3 21000 BND XIC B26:6/14 BST TON T4:35 1.0 5 0 NXB XIC T4:35/DN OTE N10:8/15 BND EOR
%   N10:30  ADS_A_INLET_PX_PSIG %
%   N7:65  HP_GAS_WRN_SP  "CONFIG Gas Inlet High Pressure Warning Setpoint" %
%   I:4.0  ADS_A_INLET_PX_READ  "PX-1" %
%   N10:33  ADS_B_INLET_PX_PSIG %
%   I:4.1  ADS_B_INLET_PX_READ  "PX-2" %
%   N10:20  OUTLET_PX_PSIG %
%   I:4.2  OUTLET_PX_READING  "PX-3" %
%   B30:0/6  INLET_PX_INSTALLED  "PX-4 Installed" %
%   N10:18  INLET_PX_PSIG %
%   I:4.3  INLET_PX_READING  "PX-4" %
%   B26:6/14  HP_GAS_WRN_EN  "CONFIG Gas Inlet High Pressure Alarm Enable" %
%   T4:35  HP_GAS_WRN_TMR  "TIMER Gas Inlet High Pressure Warning Delay" %
%   N10:8/15  HP_GAS_WARN  "WARNING Gas Inlet High Pressure" %
% Rung: 16 %
% TITLE: LOW OUTLET GAS PRESSURE %
SOR NEQ N10:0 N9:6 XIC O:2.0/4 NEQ I:4.2 21000 XIC B26:1/13 LEQ N10:20 N7:72 TON T4:94 1.0 2 0 EOR
%   N10:0  SYSTEM_STATE  "STATE The current state of the system" %
%   N9:6  SYSTEM_PURGE %
%   O:2.0/4  PURIFIED_GAS_OUT  "SV-5 OPEN" %
%   I:4.2  OUTLET_PX_READING  "PX-3" %
%   B26:1/13  LP_OUT_GAS_ALM_EN %
%   N10:20  OUTLET_PX_PSIG %
%   N7:72  LP_OUT_GAS_ALM_SP %
%   T4:94  LP_OUT_GAS_ALM_TMR %

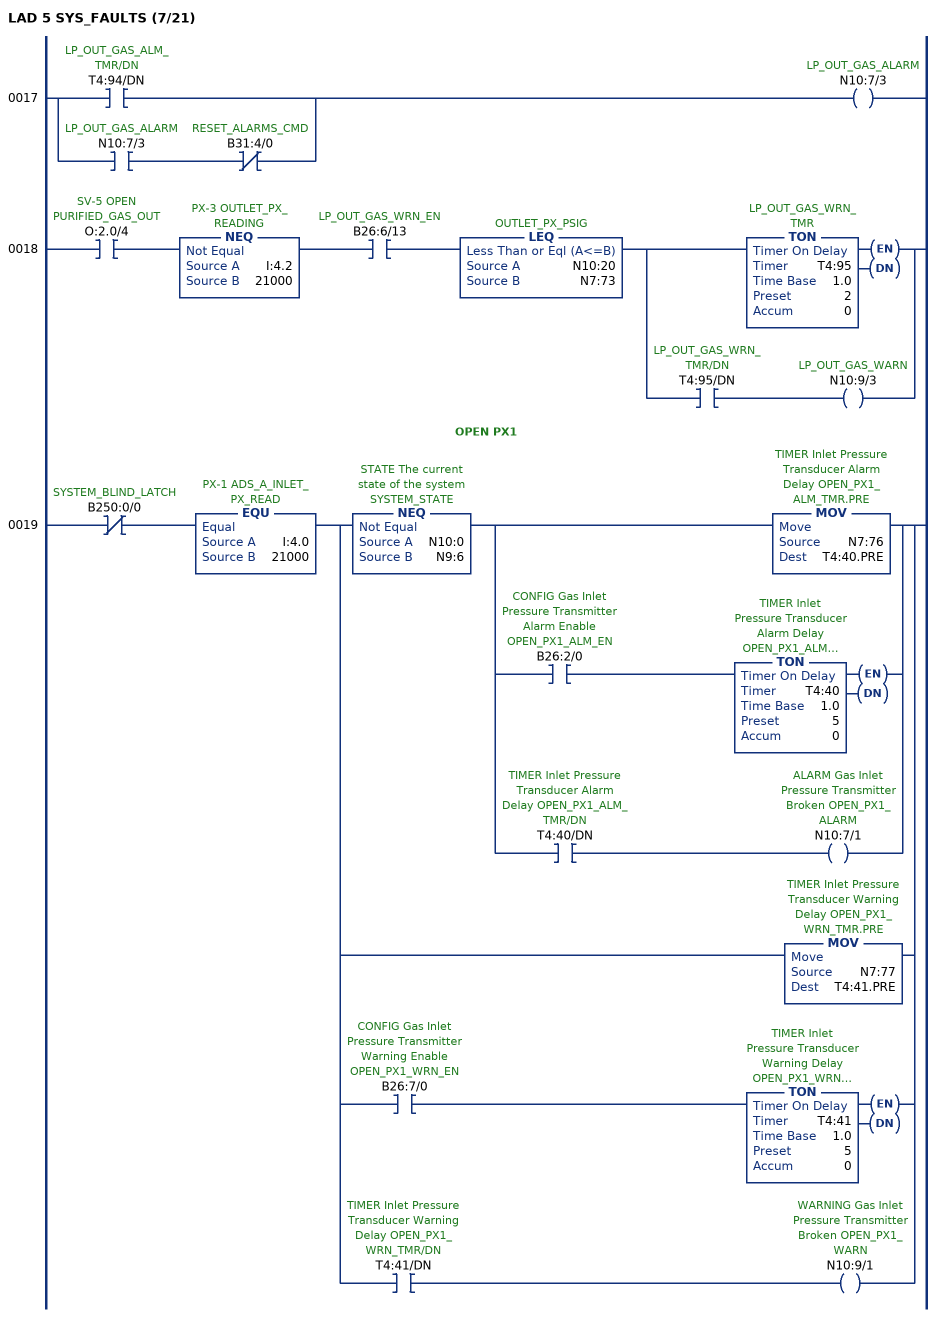
% Rung: 17 %
SOR BST XIC T4:94/DN NXB XIC N10:7/3 XIO B31:4/0 BND OTE N10:7/3 EOR
%   T4:94  LP_OUT_GAS_ALM_TMR %
%   N10:7/3  LP_OUT_GAS_ALARM %
%   B31:4/0  RESET_ALARMS_CMD %
% Rung: 18 %
SOR XIC O:2.0/4 NEQ I:4.2 21000 XIC B26:6/13 LEQ N10:20 N7:73 BST TON T4:95 1.0 2 0 NXB XIC T4:95/DN OTE N10:9/3 BND EOR
%   O:2.0/4  PURIFIED_GAS_OUT  "SV-5 OPEN" %
%   I:4.2  OUTLET_PX_READING  "PX-3" %
%   B26:6/13  LP_OUT_GAS_WRN_EN %
%   N10:20  OUTLET_PX_PSIG %
%   N7:73  LP_OUT_GAS_WRN_SP %
%   T4:95  LP_OUT_GAS_WRN_TMR %
%   N10:9/3  LP_OUT_GAS_WARN %
% Rung: 19 %
% TITLE: OPEN PX1 %
SOR XIO B250:0/0 EQU I:4.0 21000 BST NEQ N10:0 N9:6 BST MOV N7:76 T4:40.PRE NXB XIC B26:2/0 TON T4:40 1.0 5 0 NXB XIC T4:40/DN OTE N10:7/1 BND NXB BST MOV N7:77 T4:41.PRE NXB XIC B26:7/0 TON T4:41 1.0 5 0 NXB XIC T4:41/DN OTE N10:9/1 BND BND EOR
%   B250:0/0  SYSTEM_BLIND_LATCH %
%   I:4.0  ADS_A_INLET_PX_READ  "PX-1" %
%   N10:0  SYSTEM_STATE  "STATE The current state of the system" %
%   N9:6  SYSTEM_PURGE %
%   N7:76  OPEN_PX1_ALM_DLY  "CONFIG Gas Inlet Pressure Transducer Alarm Delay" %
%   T4:40  OPEN_PX1_ALM_TMR  "TIMER Inlet Pressure Transducer Alarm Delay" %
%   B26:2/0  OPEN_PX1_ALM_EN  "CONFIG Gas Inlet Pressure Transmitter Alarm Enable" %
%   N10:7/1  OPEN_PX1_ALARM  "ALARM Gas Inlet Pressure Transmitter Broken" %
%   N7:77  OPEN_PX1_WRN_DLY  "CONFIG Gas Inlet Pressure Transducer Warning Delay" %
%   T4:41  OPEN_PX1_WRN_TMR  "TIMER Inlet Pressure Transducer Warning Delay" %
%   B26:7/0  OPEN_PX1_WRN_EN  "CONFIG Gas Inlet Pressure Transmitter Warning Enable" %
%   N10:9/1  OPEN_PX1_WARN  "WARNING Gas Inlet Pressure Transmitter Broken" %

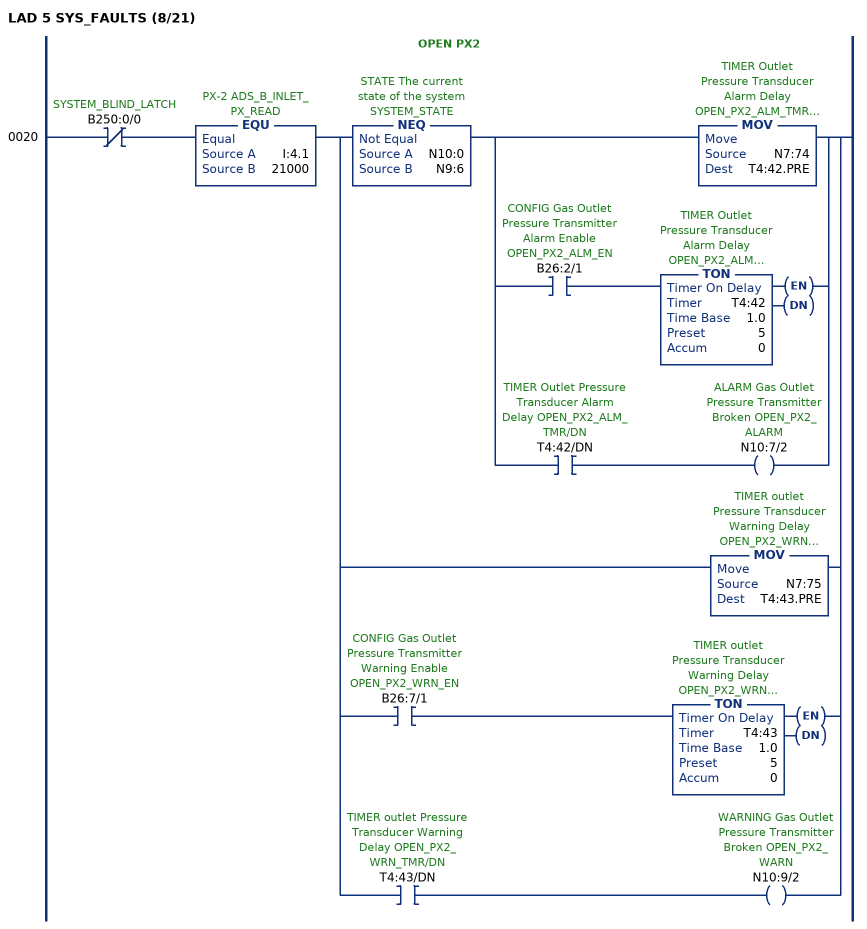
% Rung: 20 %
% TITLE: OPEN PX2 %
SOR XIO B250:0/0 EQU I:4.1 21000 BST NEQ N10:0 N9:6 BST MOV N7:74 T4:42.PRE NXB XIC B26:2/1 TON T4:42 1.0 5 0 NXB XIC T4:42/DN OTE N10:7/2 BND NXB BST MOV N7:75 T4:43.PRE NXB XIC B26:7/1 TON T4:43 1.0 5 0 NXB XIC T4:43/DN OTE N10:9/2 BND BND EOR
%   B250:0/0  SYSTEM_BLIND_LATCH %
%   I:4.1  ADS_B_INLET_PX_READ  "PX-2" %
%   N10:0  SYSTEM_STATE  "STATE The current state of the system" %
%   N9:6  SYSTEM_PURGE %
%   N7:74  OPEN_PX2_ALM_DLY  "CONFIG Gas Outlet Pressure Transducer Alarm Delay" %
%   T4:42  OPEN_PX2_ALM_TMR  "TIMER Outlet Pressure Transducer Alarm Delay" %
%   B26:2/1  OPEN_PX2_ALM_EN  "CONFIG Gas Outlet Pressure Transmitter Alarm Enable" %
%   N10:7/2  OPEN_PX2_ALARM  "ALARM Gas Outlet Pressure Transmitter Broken" %
%   N7:75  OPEN_PX2_WRN_DLY  "CONFIG Gas Outlet Pressure Transducer Warning Delay" %
%   T4:43  OPEN_PX2_WRN_TMR  "TIMER outlet Pressure Transducer Warning Delay" %
%   B26:7/1  OPEN_PX2_WRN_EN  "CONFIG Gas Outlet Pressure Transmitter Warning Enable" %
%   N10:9/2  OPEN_PX2_WARN  "WARNING Gas Outlet Pressure Transmitter Broken" %

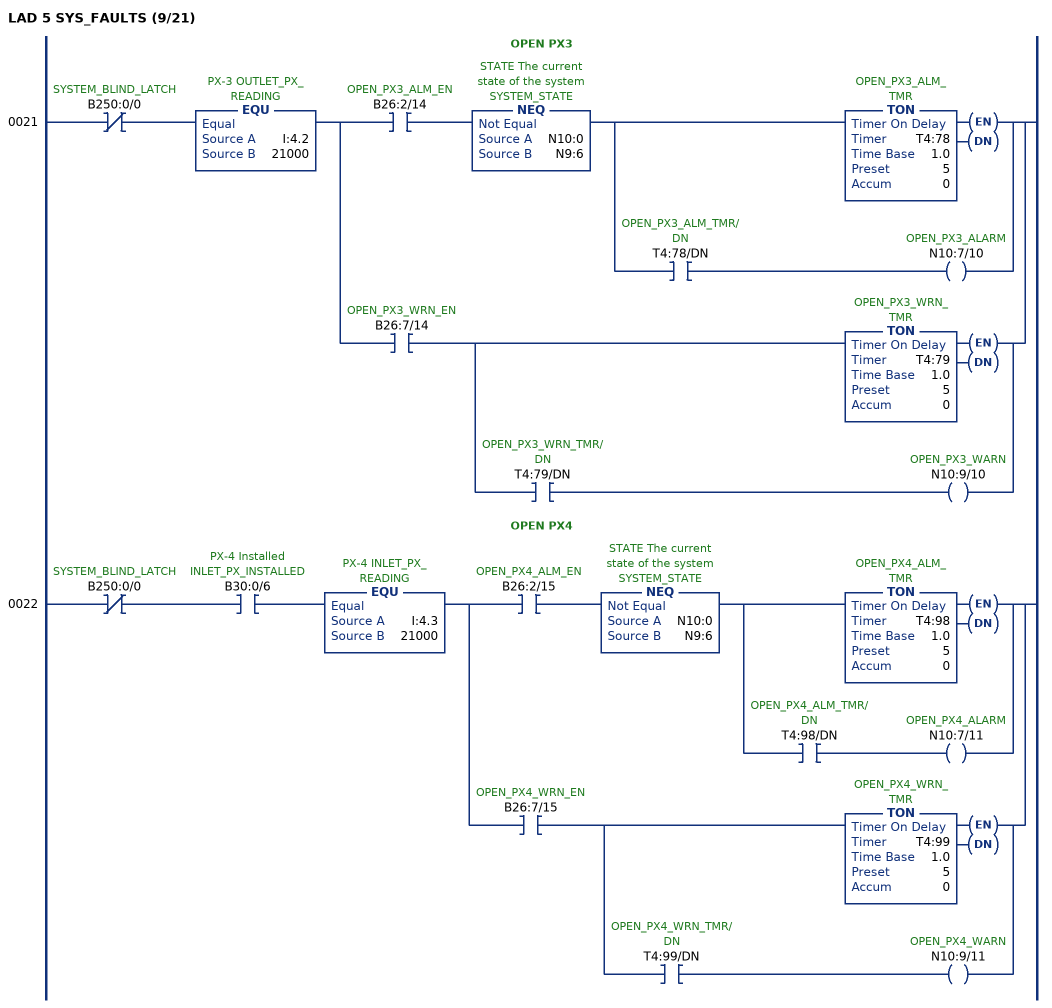
% Rung: 21 %
% TITLE: OPEN PX3 %
SOR XIO B250:0/0 EQU I:4.2 21000 BST XIC B26:2/14 NEQ N10:0 N9:6 BST TON T4:78 1.0 5 0 NXB XIC T4:78/DN OTE N10:7/10 BND NXB XIC B26:7/14 BST TON T4:79 1.0 5 0 NXB XIC T4:79/DN OTE N10:9/10 BND BND EOR
%   B250:0/0  SYSTEM_BLIND_LATCH %
%   I:4.2  OUTLET_PX_READING  "PX-3" %
%   B26:2/14  OPEN_PX3_ALM_EN %
%   N10:0  SYSTEM_STATE  "STATE The current state of the system" %
%   N9:6  SYSTEM_PURGE %
%   T4:78  OPEN_PX3_ALM_TMR %
%   N10:7/10  OPEN_PX3_ALARM %
%   B26:7/14  OPEN_PX3_WRN_EN %
%   T4:79  OPEN_PX3_WRN_TMR %
%   N10:9/10  OPEN_PX3_WARN %
% Rung: 22 %
% TITLE: OPEN PX4 %
SOR XIO B250:0/0 XIC B30:0/6 EQU I:4.3 21000 BST XIC B26:2/15 NEQ N10:0 N9:6 BST TON T4:98 1.0 5 0 NXB XIC T4:98/DN OTE N10:7/11 BND NXB XIC B26:7/15 BST TON T4:99 1.0 5 0 NXB XIC T4:99/DN OTE N10:9/11 BND BND EOR
%   B250:0/0  SYSTEM_BLIND_LATCH %
%   B30:0/6  INLET_PX_INSTALLED  "PX-4 Installed" %
%   I:4.3  INLET_PX_READING  "PX-4" %
%   B26:2/15  OPEN_PX4_ALM_EN %
%   N10:0  SYSTEM_STATE  "STATE The current state of the system" %
%   N9:6  SYSTEM_PURGE %
%   T4:98  OPEN_PX4_ALM_TMR %
%   N10:7/11  OPEN_PX4_ALARM %
%   B26:7/15  OPEN_PX4_WRN_EN %
%   T4:99  OPEN_PX4_WRN_TMR %
%   N10:9/11  OPEN_PX4_WARN %

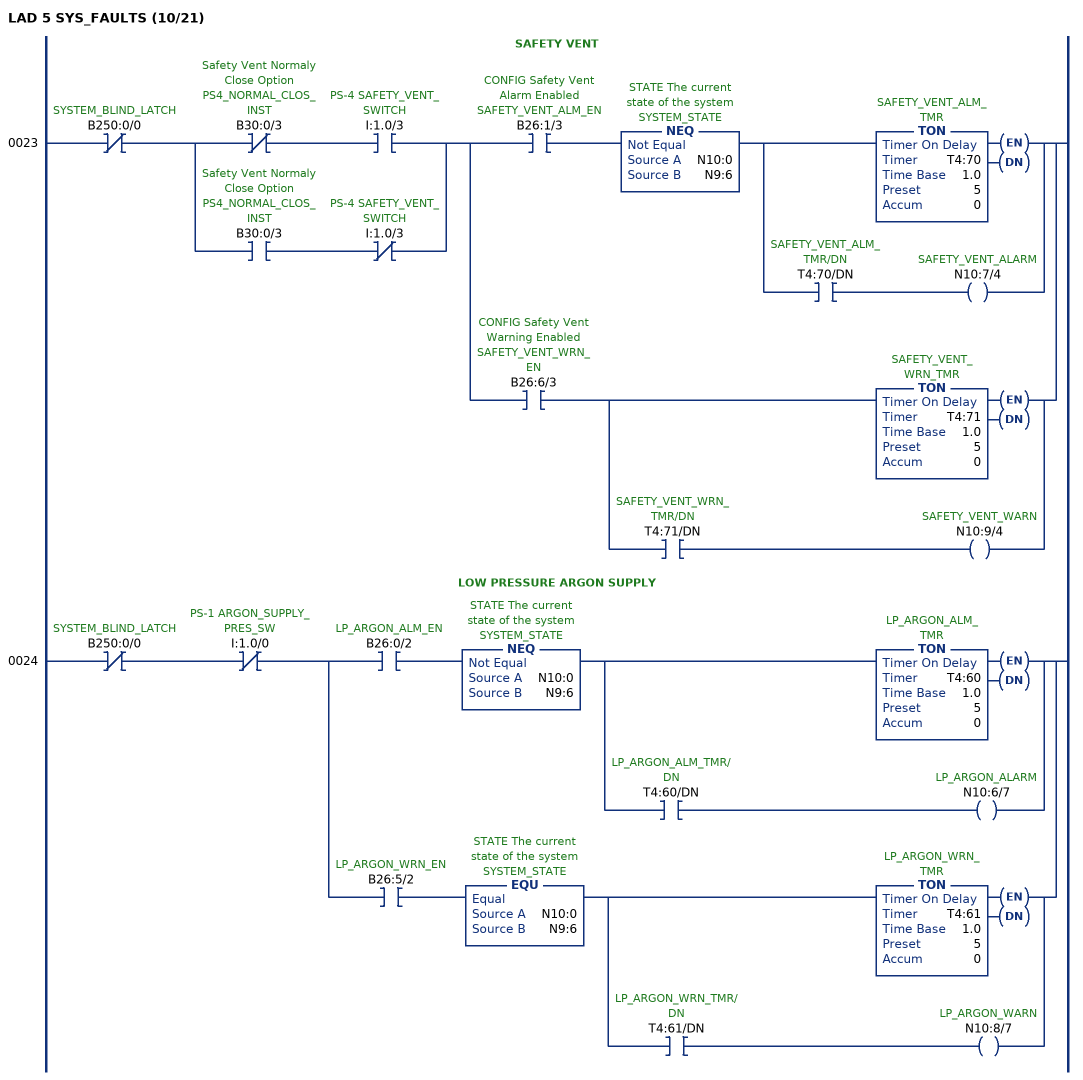
% Rung: 23 %
% TITLE: SAFETY VENT %
SOR XIO B250:0/0 BST XIO B30:0/3 XIC I:1.0/3 NXB XIC B30:0/3 XIO I:1.0/3 BND BST XIC B26:1/3 NEQ N10:0 N9:6 BST TON T4:70 1.0 5 0 NXB XIC T4:70/DN OTE N10:7/4 BND NXB XIC B26:6/3 BST TON T4:71 1.0 5 0 NXB XIC T4:71/DN OTE N10:9/4 BND BND EOR
%   B250:0/0  SYSTEM_BLIND_LATCH %
%   B30:0/3  PS4_NORMAL_CLOS_INST  "Safety Vent Normaly Close Option" %
%   I:1.0/3  SAFETY_VENT_SWITCH  "PS-4" %
%   B26:1/3  SAFETY_VENT_ALM_EN  "CONFIG Safety Vent Alarm Enabled" %
%   N10:0  SYSTEM_STATE  "STATE The current state of the system" %
%   N9:6  SYSTEM_PURGE %
%   T4:70  SAFETY_VENT_ALM_TMR %
%   N10:7/4  SAFETY_VENT_ALARM %
%   B26:6/3  SAFETY_VENT_WRN_EN  "CONFIG Safety Vent Warning Enabled" %
%   T4:71  SAFETY_VENT_WRN_TMR %
%   N10:9/4  SAFETY_VENT_WARN %
% Rung: 24 %
% TITLE: LOW PRESSURE ARGON SUPPLY %
SOR XIO B250:0/0 XIO I:1.0/0 BST XIC B26:0/2 NEQ N10:0 N9:6 BST TON T4:60 1.0 5 0 NXB XIC T4:60/DN OTE N10:6/7 BND NXB XIC B26:5/2 EQU N10:0 N9:6 BST TON T4:61 1.0 5 0 NXB XIC T4:61/DN OTE N10:8/7 BND BND EOR
%   B250:0/0  SYSTEM_BLIND_LATCH %
%   I:1.0/0  ARGON_SUPPLY_PRES_SW  "PS-1" %
%   B26:0/2  LP_ARGON_ALM_EN %
%   N10:0  SYSTEM_STATE  "STATE The current state of the system" %
%   N9:6  SYSTEM_PURGE %
%   T4:60  LP_ARGON_ALM_TMR %
%   N10:6/7  LP_ARGON_ALARM %
%   B26:5/2  LP_ARGON_WRN_EN %
%   T4:61  LP_ARGON_WRN_TMR %
%   N10:8/7  LP_ARGON_WARN %

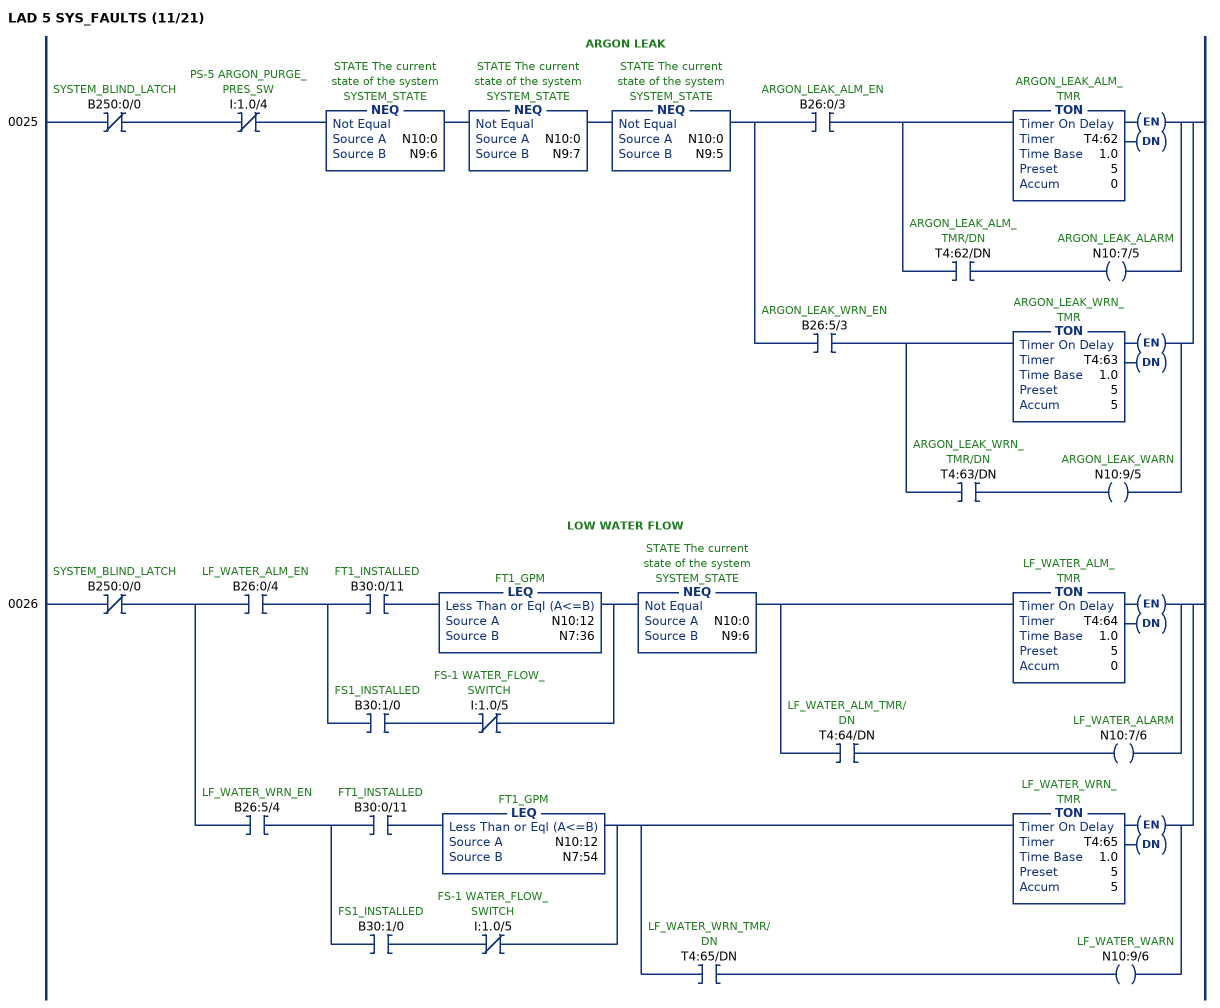
% Rung: 25 %
% TITLE: ARGON LEAK %
SOR XIO B250:0/0 XIO I:1.0/4 NEQ N10:0 N9:6 NEQ N10:0 N9:7 NEQ N10:0 N9:5 BST XIC B26:0/3 BST TON T4:62 1.0 5 0 NXB XIC T4:62/DN OTE N10:7/5 BND NXB XIC B26:5/3 BST TON T4:63 1.0 5 5 NXB XIC T4:63/DN OTE N10:9/5 BND BND EOR
%   B250:0/0  SYSTEM_BLIND_LATCH %
%   I:1.0/4  ARGON_PURGE_PRES_SW  "PS-5" %
%   N10:0  SYSTEM_STATE  "STATE The current state of the system" %
%   N9:6  SYSTEM_PURGE %
%   N9:7  SYSTEM_COLD_START %
%   N9:5  SYSTEM_QUICK_START %
%   B26:0/3  ARGON_LEAK_ALM_EN %
%   T4:62  ARGON_LEAK_ALM_TMR %
%   N10:7/5  ARGON_LEAK_ALARM %
%   B26:5/3  ARGON_LEAK_WRN_EN %
%   T4:63  ARGON_LEAK_WRN_TMR %
%   N10:9/5  ARGON_LEAK_WARN %
% Rung: 26 %
% TITLE: LOW WATER FLOW %
SOR XIO B250:0/0 BST XIC B26:0/4 BST XIC B30:0/11 LEQ N10:12 N7:36 NXB XIC B30:1/0 XIO I:1.0/5 BND NEQ N10:0 N9:6 BST TON T4:64 1.0 5 0 NXB XIC T4:64/DN OTE N10:7/6 BND NXB XIC B26:5/4 BST XIC B30:0/11 LEQ N10:12 N7:54 NXB XIC B30:1/0 XIO I:1.0/5 BND BST TON T4:65 1.0 5 5 NXB XIC T4:65/DN OTE N10:9/6 BND BND EOR
%   B250:0/0  SYSTEM_BLIND_LATCH %
%   B26:0/4  LF_WATER_ALM_EN %
%   B30:0/11  FT1_INSTALLED %
%   N10:12  FT1_GPM %
%   N7:36  LF_WATER_ALM_SP %
%   B30:1/0  FS1_INSTALLED %
%   I:1.0/5  WATER_FLOW_SWITCH  "FS-1" %
%   N10:0  SYSTEM_STATE  "STATE The current state of the system" %
%   N9:6  SYSTEM_PURGE %
%   T4:64  LF_WATER_ALM_TMR %
%   N10:7/6  LF_WATER_ALARM %
%   B26:5/4  LF_WATER_WRN_EN %
%   N7:54  LF_WATER_WRN_SP %
%   T4:65  LF_WATER_WRN_TMR %
%   N10:9/6  LF_WATER_WARN %

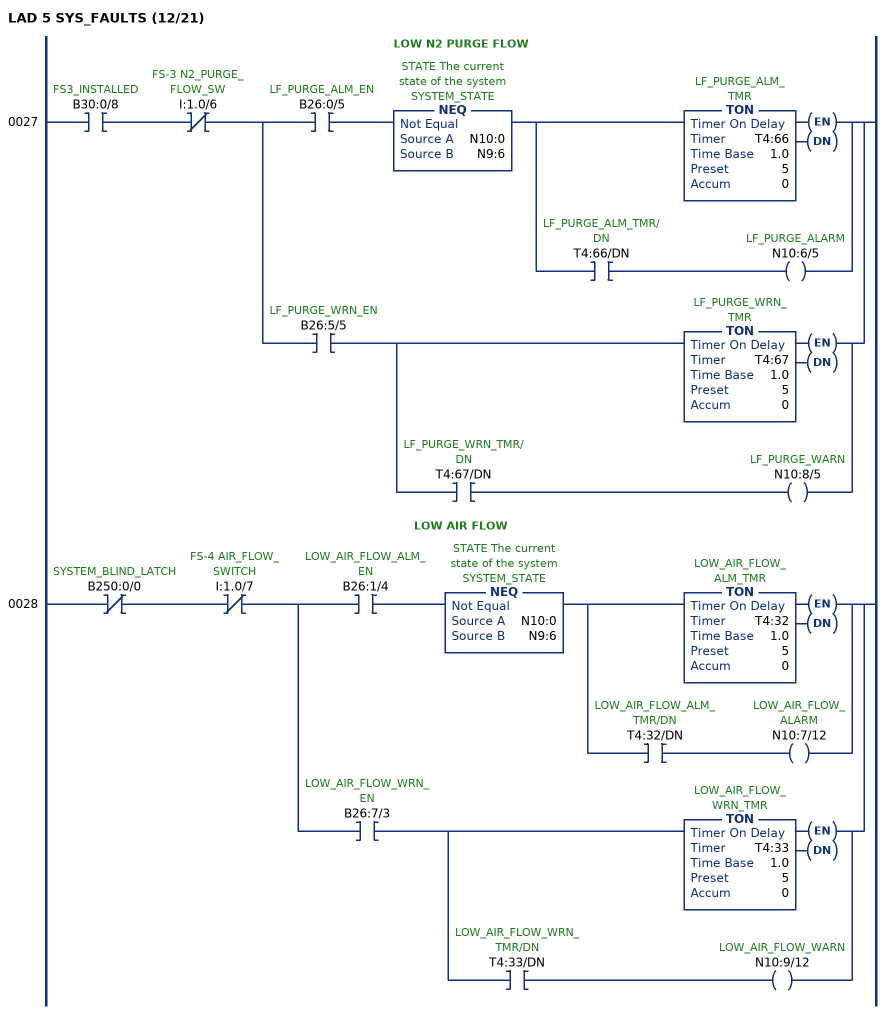
% Rung: 27 %
% TITLE: LOW N2 PURGE FLOW %
SOR XIC B30:0/8 XIO I:1.0/6 BST XIC B26:0/5 NEQ N10:0 N9:6 BST TON T4:66 1.0 5 0 NXB XIC T4:66/DN OTE N10:6/5 BND NXB XIC B26:5/5 BST TON T4:67 1.0 5 0 NXB XIC T4:67/DN OTE N10:8/5 BND BND EOR
%   B30:0/8  FS3_INSTALLED %
%   I:1.0/6  N2_PURGE_FLOW_SW  "FS-3" %
%   B26:0/5  LF_PURGE_ALM_EN %
%   N10:0  SYSTEM_STATE  "STATE The current state of the system" %
%   N9:6  SYSTEM_PURGE %
%   T4:66  LF_PURGE_ALM_TMR %
%   N10:6/5  LF_PURGE_ALARM %
%   B26:5/5  LF_PURGE_WRN_EN %
%   T4:67  LF_PURGE_WRN_TMR %
%   N10:8/5  LF_PURGE_WARN %
% Rung: 28 %
% TITLE: LOW AIR FLOW %
SOR XIO B250:0/0 XIO I:1.0/7 BST XIC B26:1/4 NEQ N10:0 N9:6 BST TON T4:32 1.0 5 0 NXB XIC T4:32/DN OTE N10:7/12 BND NXB XIC B26:7/3 BST TON T4:33 1.0 5 0 NXB XIC T4:33/DN OTE N10:9/12 BND BND EOR
%   B250:0/0  SYSTEM_BLIND_LATCH %
%   I:1.0/7  AIR_FLOW_SWITCH  "FS-4" %
%   B26:1/4  LOW_AIR_FLOW_ALM_EN %
%   N10:0  SYSTEM_STATE  "STATE The current state of the system" %
%   N9:6  SYSTEM_PURGE %
%   T4:32  LOW_AIR_FLOW_ALM_TMR %
%   N10:7/12  LOW_AIR_FLOW_ALARM %
%   B26:7/3  LOW_AIR_FLOW_WRN_EN %
%   T4:33  LOW_AIR_FLOW_WRN_TMR %
%   N10:9/12  LOW_AIR_FLOW_WARN %

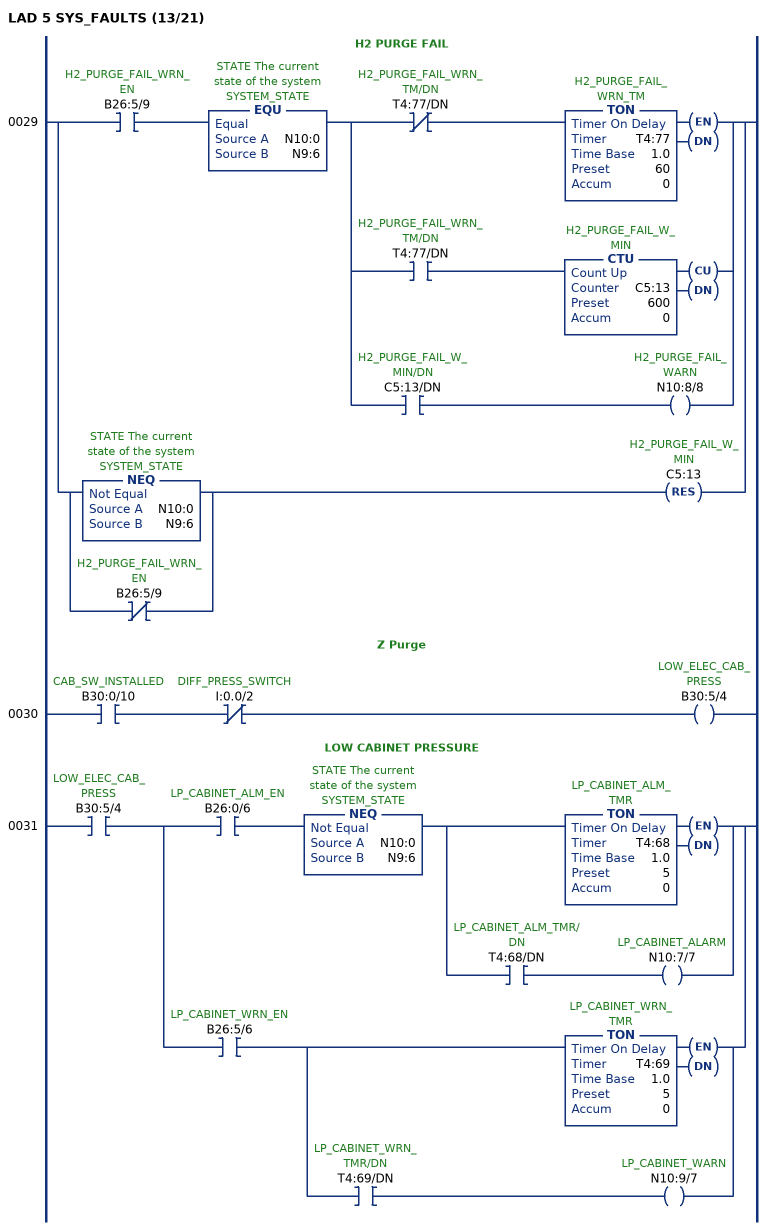
% Rung: 29 %
% TITLE: H2 PURGE FAIL %
SOR BST XIC B26:5/9 EQU N10:0 N9:6 BST XIO T4:77/DN TON T4:77 1.0 60 0 NXB XIC T4:77/DN CTU C5:13 600 0 NXB XIC C5:13/DN OTE N10:8/8 BND NXB BST NEQ N10:0 N9:6 NXB XIO B26:5/9 BND RES C5:13 BND EOR
%   B26:5/9  H2_PURGE_FAIL_WRN_EN %
%   N10:0  SYSTEM_STATE  "STATE The current state of the system" %
%   N9:6  SYSTEM_PURGE %
%   T4:77  H2_PURGE_FAIL_WRN_TM %
%   C5:13  H2_PURGE_FAIL_W_MIN %
%   N10:8/8  H2_PURGE_FAIL_WARN %
% Rung: 30 %
% TITLE: Z Purge %
SOR XIC B30:0/10 XIO I:0.0/2 OTE B30:5/4 EOR
%   B30:0/10  CAB_SW_INSTALLED %
%   I:0.0/2  DIFF_PRESS_SWITCH %
%   B30:5/4  LOW_ELEC_CAB_PRESS %
% Rung: 31 %
% TITLE: LOW CABINET PRESSURE %
SOR XIC B30:5/4 BST XIC B26:0/6 NEQ N10:0 N9:6 BST TON T4:68 1.0 5 0 NXB XIC T4:68/DN OTE N10:7/7 BND NXB XIC B26:5/6 BST TON T4:69 1.0 5 0 NXB XIC T4:69/DN OTE N10:9/7 BND BND EOR
%   B30:5/4  LOW_ELEC_CAB_PRESS %
%   B26:0/6  LP_CABINET_ALM_EN %
%   N10:0  SYSTEM_STATE  "STATE The current state of the system" %
%   N9:6  SYSTEM_PURGE %
%   T4:68  LP_CABINET_ALM_TMR %
%   N10:7/7  LP_CABINET_ALARM %
%   B26:5/6  LP_CABINET_WRN_EN %
%   T4:69  LP_CABINET_WRN_TMR %
%   N10:9/7  LP_CABINET_WARN %

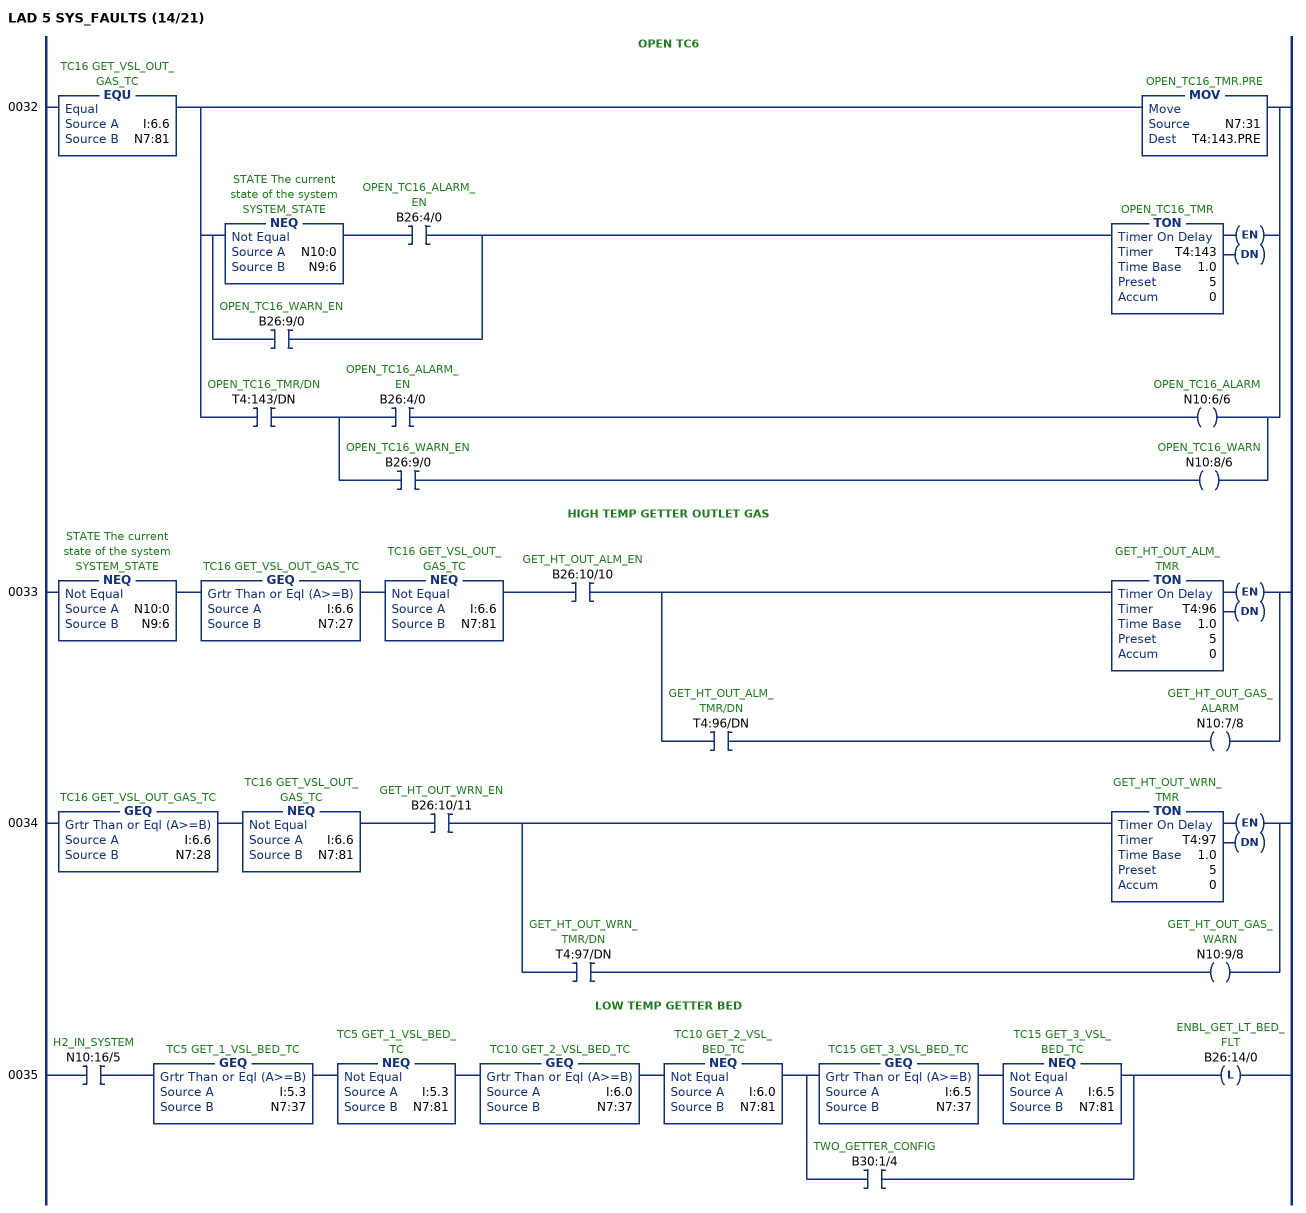
% Rung: 32 %
% TITLE: OPEN TC6 %
SOR EQU I:6.6 N7:81 BST MOV N7:31 T4:143.PRE NXB BST NEQ N10:0 N9:6 XIC B26:4/0 NXB XIC B26:9/0 BND TON T4:143 1.0 5 0 NXB XIC T4:143/DN BST XIC B26:4/0 OTE N10:6/6 NXB XIC B26:9/0 OTE N10:8/6 BND BND EOR
%   I:6.6  GET_VSL_OUT_GAS_TC  "TC16" %
%   N7:81  TC_OPEN_SP  "CONFIG The value read by an open TC input" %
%   N7:31  OPEN_TC_DLY %
%   T4:143  OPEN_TC16_TMR %
%   N10:0  SYSTEM_STATE  "STATE The current state of the system" %
%   N9:6  SYSTEM_PURGE %
%   B26:4/0  OPEN_TC16_ALARM_EN %
%   B26:9/0  OPEN_TC16_WARN_EN %
%   N10:6/6  OPEN_TC16_ALARM %
%   N10:8/6  OPEN_TC16_WARN %
% Rung: 33 %
% TITLE: HIGH TEMP GETTER OUTLET GAS %
SOR NEQ N10:0 N9:6 GEQ I:6.6 N7:27 NEQ I:6.6 N7:81 XIC B26:10/10 BST TON T4:96 1.0 5 0 NXB XIC T4:96/DN OTE N10:7/8 BND EOR
%   N10:0  SYSTEM_STATE  "STATE The current state of the system" %
%   N9:6  SYSTEM_PURGE %
%   I:6.6  GET_VSL_OUT_GAS_TC  "TC16" %
%   N7:27  GET_HT_OUT_ALM_SP %
%   N7:81  TC_OPEN_SP  "CONFIG The value read by an open TC input" %
%   B26:10/10  GET_HT_OUT_ALM_EN %
%   T4:96  GET_HT_OUT_ALM_TMR %
%   N10:7/8  GET_HT_OUT_GAS_ALARM %
% Rung: 34 %
SOR GEQ I:6.6 N7:28 NEQ I:6.6 N7:81 XIC B26:10/11 BST TON T4:97 1.0 5 0 NXB XIC T4:97/DN OTE N10:9/8 BND EOR
%   I:6.6  GET_VSL_OUT_GAS_TC  "TC16" %
%   N7:28  GET_HT_OUT_WRN_SP %
%   N7:81  TC_OPEN_SP  "CONFIG The value read by an open TC input" %
%   B26:10/11  GET_HT_OUT_WRN_EN %
%   T4:97  GET_HT_OUT_WRN_TMR %
%   N10:9/8  GET_HT_OUT_GAS_WARN %
% Rung: 35 %
% TITLE: LOW TEMP GETTER BED %
SOR XIC N10:16/5 GEQ I:5.3 N7:37 NEQ I:5.3 N7:81 GEQ I:6.0 N7:37 NEQ I:6.0 N7:81 BST GEQ I:6.5 N7:37 NEQ I:6.5 N7:81 NXB XIC B30:1/4 BND OTL B26:14/0 EOR
%   N10:16/5  H2_IN_SYSTEM %
%   I:5.3  GET_1_VSL_BED_TC  "TC5" %
%   N7:37  GET_LT_SHUTDOWN_SP %
%   N7:81  TC_OPEN_SP  "CONFIG The value read by an open TC input" %
%   I:6.0  GET_2_VSL_BED_TC  "TC10" %
%   I:6.5  GET_3_VSL_BED_TC  "TC15" %
%   B30:1/4  TWO_GETTER_CONFIG %
%   B26:14/0  ENBL_GET_LT_BED_FLT %

